// TwinCAT 3 PLC project MAIN
// ProgramVersion: 3.1.4024.0
// CompilerDefines: VISU_USEWSTRING
// libraries:
//   VisuElemMeter, * (System)
//   Tc2_EtherCAT, * (Beckhoff Automation GmbH)
//   Tc2_ModbusRTU, * (Beckhoff Automation GmbH)
//   Tc2_Standard, * (Beckhoff Automation GmbH)
//   Tc2_SUPS, * (Beckhoff Automation GmbH)
//   Tc2_System, * (Beckhoff Automation GmbH)
//   Tc2_Utilities, * (Beckhoff Automation GmbH)
//   Tc3_EventLogger, * (Beckhoff Automation GmbH)
//   Tc3_Module, * (Beckhoff Automation GmbH)
//   VisuDialogs, * (System)
// project tree:
//   DUTs/ ST_4Bytes.TcDUT, ST_Error.TcDUT, U_4Bytes2Real.TcDUT
//   / GlobalTextList.TcGTLO, ImagePool.TcIPO (not stored), PlcTask.TcTTO, PlcTask2.TcTTO, RecipeManager.TcRMO (not stored), Visualization Manager.TcVMO (not stored), VISU_TASK.TcTTO
//   GVLs/ GVL.TcGVL, GVL_ADS.TcGVL, GVL_HMI.TcGVL, GVL_IO.TcGVL, GVL_IoT.TcGVL, GVL_OF_VU.TcGVL, GVL_Retain.TcGVL
//   POUs/Components/Child Components/ FB_Conveyor.TcPOU, FB_Cylinder.TcPOU, FB_Interface_EtherCat.TcPOU, FB_Interface_MbRtu.TcPOU, FB_Inverter.TcPOU, FB_Loadcell.TcPOU, FB_SuctionCup.TcPOU
//   POUs/Components/Interfaces/ I_Conveyor.TcIO, I_Cylinder.TcIO, I_Inverter.TcIO, I_LoadCell.TcIO, I_SuctionCup.TcIO
//   POUs/Components/Sim Components/ FB_Conveyor_Sim.TcPOU, FB_Cylinder_Sim.TcPOU, FB_Inverter_Sim.TcPOU, FB_LoadCell_Sim.TcPOU, FB_SuctionCup_Sim.TcPOU
//   POUs/Functions/ FB_EventButton.TcPOU, FB_Eventlogger.TcPOU, F_SetError.TcPOU, F_SetWarning.TcPOU
//   POUs/Machines/ PR_Conveyor_Out.TcPOU, PR_Line01.TcPOU, PR_Line02.TcPOU
//   POUs/ MAIN.TcPOU, MAIN_LINE2.TcPOU
//   POUs/Modules/ FB_CupSupplyModule.TcPOU, FB_FoodMixerModule.TcPOU, FB_FoodWeightModule.TcPOU, FB_LidCloseModule.TcPOU, FB_LidSupplyModule.TcPOU, FB_Transfer.TcPOU, FB_WormWeightModule.TcPOU
//   POUs/Recipe/ PRG_MainRecipe1.TcPOU, PRG_MainRecipe1_1.TcPOU, PRG_RecipeList1.TcPOU, PRG_RecipeList1_1.TcPOU
//   VISUs/Alarm/ N_Alarm.TcVIS, N_Alarm_1.TcVIS
//   VISUs/IO/ N_Parameter_1.TcVIS, N_Parameter_2.TcVIS, N_PLC_I1.TcVIS, N_PLC_I1_next.TcVIS, N_PLC_I2.TcVIS, N_PLC_I2_next.TcVIS, N_PLC_O1.TcVIS, N_PLC_O2.TcVIS
//   VISUs/Main_Line/ MAIN_LINE1.TcVIS, MAIN_LINE2.TcVIS
//   VISUs/Manual/Line1/ N_FoodSupply1.TcVIS, N_JarSupply1.TcVIS, N_LidPressing1.TcVIS, N_LidSupply1.TcVIS, N_Tranfer1.TcVIS, N_WormWeight1.TcVIS
//   VISUs/Manual/Line2/ N_FoodSupply2.TcVIS, N_JarSupply2.TcVIS, N_LidPressing2.TcVIS, N_LidSupply2.TcVIS, N_Tranfer2.TcVIS, N_WormWeight2.TcVIS
//   VISUs/Recipe/ N_Recipe_Line1.TcVIS, N_Recipe_Line2.TcVIS
//   VISUs/Setting/ N_Setting_Delay_FoodSupply1.TcVIS, N_Setting_Delay_FoodSupply2.TcVIS, N_Setting_Delay_JarSupply1.TcVIS, N_Setting_Delay_JarSupply2.TcVIS, N_Setting_Delay_LidPressing1.TcVIS, N_Setting_Delay_LidPressing2.TcVIS, N_Setting_Delay_LidSupply1.TcVIS, N_Setting_Delay_LidSupply2.TcVIS, N_Setting_Delay_Tranfer1.TcVIS, N_Setting_Delay_Tranfer2.TcVIS, N_Setting_Delay_WormWeight1.TcVIS, N_Setting_Delay_WorwWeight2.TcVIS, N_Setting_Line1.TcVIS, N_Setting_Line2.TcVIS
//   VISUs/Title/ N_Footer_Alarm.TcVIS, N_Footer_Alarm_1.TcVIS, N_Footer_Line1.TcVIS, N_Footer_Line2.TcVIS, N_Header.TcVIS, N_Login.TcVIS, startpage.TcVIS
// real-time tasks:
//   TASK PlcTask: cycle T#10ms, priority 20, ADS port 350
//   TASK VISU_TASK: cycle T#10ms, priority 30, ADS port 351
//   TASK PlcTask2: cycle T#10ms, priority 21, ADS port 352
//   TASK VISU_TASK1: cycle T#10ms, priority 1, ADS port 353
// I/O:
//   DEVICE Device 1 (EtherCAT) (disabled), AmsNetId 192.168.1.12.2.1
//     Term 1 (EK1200) [EK1200-5000 EtherCAT Power supply (2A E-Bus)]
//       Term 2 (EL1008) [EL1008 8Ch. Dig. Input 24V, 3ms]
//       Term 3 (EL1008) [EL1008 8Ch. Dig. Input 24V, 3ms]
//       Term 4 (EL1008) [EL1008 8Ch. Dig. Input 24V, 3ms]
//       Term 5 (EL1008) [EL1008 8Ch. Dig. Input 24V, 3ms]
//       Term 6 (EL1008) [EL1008 8Ch. Dig. Input 24V, 3ms]
//       Term 7 (EL1008) [EL1008 8Ch. Dig. Input 24V, 3ms]
//       Term 8 (EL1819) [EL1819 16Ch. Dig. Input 24V, 10µs]
//       Term 9 (EL2809) [EL2809 16Ch. Dig. Output 24V, 0.5A]
//       Term 10 (EL2809) [EL2809 16Ch. Dig. Output 24V, 0.5A]
//       Term 11 (EL2809-0015) [EL2809-0015 16Ch. Dig. Output 24V DC, 0.35A, not short-circuit proof]
//       Term 12 (EL6021) [EL6021 Interface (RS422/485)]
//       Term 13 (EK1110) [EK1110 EtherCAT extension]
//     Box 14 (TLBETHERCAT) [TLBETHERCAT]
//     Box 15 (TLBETHERCAT) [TLBETHERCAT]
//     Box 16 (IND360) [IND360 ECS]
//     Box 17 (IND360) [IND360 ECS]
//   DEVICE Device 3 (NOV-DP-RAM) (disabled)
// variable links:
//   MAIN/MAIN Instance <-> Device 1 (EtherCAT)/Box 14 (TLBETHERCAT)
//     PlcTask2 Inputs/PR_Line02.fb_WormWeight.fbLoadcell.fbInterface.StatusLaumas1 <-> TxPDO/1 Byte In (13)
//     PlcTask2 Inputs/PR_Line02.fb_WormWeight.fbLoadcell.fbInterface.StatusLaumas2 <-> TxPDO/1 Byte In (12)
//     PlcTask2 Inputs/PR_Line02.fb_WormWeight.fbLoadcell.fbInterface.WeightLaumas1 <-> TxPDO/1 Byte In (3)
//     PlcTask2 Inputs/PR_Line02.fb_WormWeight.fbLoadcell.fbInterface.WeightLaumas2 <-> TxPDO/1 Byte In (2)
//     PlcTask2 Inputs/PR_Line02.fb_WormWeight.fbLoadcell.fbInterface.WeightLaumas3 <-> TxPDO/1 Byte In (1)
//     PlcTask2 Inputs/PR_Line02.fb_WormWeight.fbLoadcell.fbInterface.WeightLaumas4 <-> TxPDO/1 Byte In (0)
//     PlcTask2 Outputs/PR_Line02.fb_WormWeight.fbLoadcell.fbInterface.CMDLaumas <-> RxPDO/1 Byte Out (1)
//   MAIN/MAIN Instance <-> Device 1 (EtherCAT)/Box 15 (TLBETHERCAT)
//     PlcTask2 Inputs/PR_Line02.fb_FoodWeight.fbLoadcell.fbInterface.StatusLaumas1 <-> TxPDO/1 Byte In (13)
//     PlcTask2 Inputs/PR_Line02.fb_FoodWeight.fbLoadcell.fbInterface.StatusLaumas2 <-> TxPDO/1 Byte In (12)
//     PlcTask2 Inputs/PR_Line02.fb_FoodWeight.fbLoadcell.fbInterface.WeightLaumas1 <-> TxPDO/1 Byte In (3)
//     PlcTask2 Inputs/PR_Line02.fb_FoodWeight.fbLoadcell.fbInterface.WeightLaumas2 <-> TxPDO/1 Byte In (2)
//     PlcTask2 Inputs/PR_Line02.fb_FoodWeight.fbLoadcell.fbInterface.WeightLaumas3 <-> TxPDO/1 Byte In (1)
//     PlcTask2 Inputs/PR_Line02.fb_FoodWeight.fbLoadcell.fbInterface.WeightLaumas4 <-> TxPDO/1 Byte In (0)
//     PlcTask2 Outputs/PR_Line02.fb_FoodWeight.fbLoadcell.fbInterface.CMDLaumas <-> RxPDO/1 Byte Out (1)
//   MAIN/MAIN Instance <-> Device 1 (EtherCAT)/Box 16 (IND360)
//     PlcTask Inputs/PR_Line01.fb_WormWeight.fbLoadcell.fbInterface.IND_M_RD_Float <-> TxPDO-2Block/MB1 Requested Measuring Value
//     PlcTask Inputs/PR_Line01.fb_WormWeight.fbLoadcell.fbInterface.IND_M_RD_Response <-> TxPDO-2Block/MB1 Response
//     PlcTask Inputs/PR_Line01.fb_WormWeight.fbLoadcell.fbInterface.IND_M_RD_Status <-> TxPDO-2Block/MB1 Scale Status
//     PlcTask Inputs/PR_Line01.fb_WormWeight.fbLoadcell.fbInterface.IND_SB_STT1 <-> TxPDO-2Block/SB1 Status Group 1
//     PlcTask Inputs/PR_Line01.fb_WormWeight.fbLoadcell.fbInterface.IND_SB_STT2 <-> TxPDO-2Block/SB1 Status Group 2
//     PlcTask Inputs/PR_Line01.fb_WormWeight.fbLoadcell.fbInterface.IND_SB_STT3 <-> TxPDO-2Block/SB1 Status Group 3
//     PlcTask Outputs/PR_Line01.fb_WormWeight.fbLoadcell.fbInterface.IND_M_WR_Command <-> RxPDO-2Block/MB1 Command
//     PlcTask Outputs/PR_Line01.fb_WormWeight.fbLoadcell.fbInterface.IND_M_WR_Float <-> RxPDO-2Block/MB1 Command Value
//   MAIN/MAIN Instance <-> Device 1 (EtherCAT)/Box 17 (IND360)
//     PlcTask Inputs/PR_Line01.fb_FoodWeight.fbLoadcell.fbInterface.IND_M_RD_Float <-> TxPDO-2Block/MB1 Requested Measuring Value
//     PlcTask Inputs/PR_Line01.fb_FoodWeight.fbLoadcell.fbInterface.IND_M_RD_Response <-> TxPDO-2Block/MB1 Response
//     PlcTask Inputs/PR_Line01.fb_FoodWeight.fbLoadcell.fbInterface.IND_M_RD_Status <-> TxPDO-2Block/MB1 Scale Status
//     PlcTask Inputs/PR_Line01.fb_FoodWeight.fbLoadcell.fbInterface.IND_SB_STT1 <-> TxPDO-2Block/SB1 Status Group 1
//     PlcTask Inputs/PR_Line01.fb_FoodWeight.fbLoadcell.fbInterface.IND_SB_STT2 <-> TxPDO-2Block/SB1 Status Group 2
//     PlcTask Inputs/PR_Line01.fb_FoodWeight.fbLoadcell.fbInterface.IND_SB_STT3 <-> TxPDO-2Block/SB1 Status Group 3
//     PlcTask Outputs/PR_Line01.fb_FoodWeight.fbLoadcell.fbInterface.IND_M_WR_Command <-> RxPDO-2Block/MB1 Command
//     PlcTask Outputs/PR_Line01.fb_FoodWeight.fbLoadcell.fbInterface.IND_M_WR_Float <-> RxPDO-2Block/MB1 Command Value
//   MAIN/MAIN Instance <-> Device 1 (EtherCAT)/Term 1 (EK1200)/Term 10 (EL2809)
//     PlcTask Outputs/PR_Line01.fb_CupSupply.fbCylinder_Dw.bMoveRetract <-> Channel 9/Output
//     PlcTask Outputs/PR_Line01.fb_CupSupply.fbCylinder_Suction.bMoveRetract <-> Channel 14/Output
//     PlcTask Outputs/PR_Line01.fb_CupSupply.fbCylinder_Up.bMoveExtend <-> Channel 8/Output
//     PlcTask Outputs/PR_Line01.fb_LidClose.fbCylinder_LidClose.bMoveExtend <-> Channel 15/Output
//     PlcTask Outputs/PR_Line01.fb_LidSupply.fbCylinder_LidStopper.bMoveRetract <-> Channel 11/Output
//     PlcTask Outputs/PR_Line01.fb_LidSupply.fbCylinder_Suction.bMoveExtend <-> Channel 12/Output
//     PlcTask Outputs/PR_Line01.fb_LidSupply.fbLidSuctionValve.bSuck <-> Channel 13/Output
//     PlcTask Outputs/PR_Line01.fb_Transfer.fbCylinder_Clip.bMoveRetract <-> Channel 16/Output
//     PlcTask Outputs/PR_Line01.fb_WormWeight.fbCylinder.bMoveRetract <-> Channel 10/Output
//     PlcTask2 Outputs/PR_Line02.fb_CupSupply.fbCylinder_Suction.bMoveRetract <-> Channel 3/Output
//     PlcTask2 Outputs/PR_Line02.fb_LidClose.fbCylinder_LidClose.bMoveExtend <-> Channel 4/Output
//     PlcTask2 Outputs/PR_Line02.fb_LidSupply.fbCylinder_Suction.bMoveExtend <-> Channel 1/Output
//     PlcTask2 Outputs/PR_Line02.fb_LidSupply.fbLidSuctionValve.bSuck <-> Channel 2/Output
//     PlcTask2 Outputs/PR_Line02.fb_Transfer.fbCylinder_Clip.bMoveRetract <-> Channel 5/Output
//     PlcTask2 Outputs/PR_Line02.fb_Transfer.fbCylinder_Comb.bMoveExtend <-> Channel 6/Output
//     PlcTask2 Outputs/PR_Line02.fb_Transfer.fbCylinder_Move_Comb.bMoveExtend <-> Channel 7/Output
//   MAIN/MAIN Instance <-> Device 1 (EtherCAT)/Term 1 (EK1200)/Term 11 (EL2809-0015)
//     PlcTask Outputs/PR_Line01.fb_FoodMixer.fbInverter.bReverse <-> Channel 3/Output
//     PlcTask Outputs/PR_Line01.fb_FoodWeight.fbDriver.bReverse <-> Channel 6/Output
//     PlcTask Outputs/PR_Line01.fb_Transfer.fbCylinder_Comb.bMoveExtend <-> Channel 1/Output
//     PlcTask Outputs/PR_Line01.fb_Transfer.fbCylinder_Move_Comb.bMoveExtend <-> Channel 2/Output
//     PlcTask2 Outputs/PR_Line02.fb_FoodMixer.fbInverter.bReverse <-> Channel 4/Output
//     PlcTask2 Outputs/PR_Line02.fb_FoodWeight.fbDriver.bReverse <-> Channel 5/Output
//   MAIN/MAIN Instance <-> Device 1 (EtherCAT)/Term 1 (EK1200)/Term 12 (EL6021)
//     PlcTask Inputs/GVL.fbModbus.InData/D[{0..21}] <-> COM TxPDO-Map Inputs/Data In {0..21}  (22 links)
//     PlcTask Inputs/GVL.fbModbus.InData/Status <-> COM TxPDO-Map Inputs/Status
//     PlcTask Outputs/GVL.fbModbus.OutData/Ctrl <-> COM RxPDO-Map Outputs/Ctrl
//     PlcTask Outputs/GVL.fbModbus.OutData/D[{0..21}] <-> COM RxPDO-Map Outputs/Data Out {0..21}  (22 links)
//   MAIN/MAIN Instance <-> Device 1 (EtherCAT)/Term 1 (EK1200)/Term 2 (EL1008)
//     PlcTask Inputs/GVL_IO.bEmer <-> Channel 4/Input
//     PlcTask Inputs/GVL_IO.bReset <-> Channel 3/Input
//     PlcTask Inputs/GVL_IO.bStart <-> Channel 1/Input
//     PlcTask Inputs/GVL_IO.bStop <-> Channel 2/Input
//     PlcTask Inputs/PR_Conveyor_Out.fb_Conveyor.bError_Motor_Mixer <-> Channel 7/Input
//     PlcTask Inputs/PR_Line01.fb_FoodMixer.bError_Motor_Mixer <-> Channel 8/Input
//     PlcTask2 Inputs/PR_Line02.fb_FoodMixer.bError_Motor_Mixer <-> Channel 5/Input
//     PlcTask2 Inputs/PR_Line02.fb_WormWeight.bError_Inverter <-> Channel 6/Input
//   MAIN/MAIN Instance <-> Device 1 (EtherCAT)/Term 1 (EK1200)/Term 3 (EL1008)
//     PlcTask Inputs/PR_Line01.fb_FoodWeight.bError_Driver <-> Channel 3/Input
//     PlcTask Inputs/PR_Line01.fb_WormWeight.bError_Inverter <-> Channel 1/Input
//     PlcTask2 Inputs/PR_Line02.fb_CupSupply.bCupDrop <-> Channel 8/Input
//     PlcTask2 Inputs/PR_Line02.fb_CupSupply.bCupEmpty <-> Channel 4/Input
//     PlcTask2 Inputs/PR_Line02.fb_CupSupply.fbCylinder_Dw.bAtExtend <-> Channel 7/Input
//     PlcTask2 Inputs/PR_Line02.fb_CupSupply.fbCylinder_Dw.bAtRetract <-> Channel 6/Input
//     PlcTask2 Inputs/PR_Line02.fb_CupSupply.fbCylinder_Up.bAtRetract <-> Channel 5/Input
//     PlcTask2 Inputs/PR_Line02.fb_FoodWeight.bError_Driver <-> Channel 2/Input
//   MAIN/MAIN Instance <-> Device 1 (EtherCAT)/Term 1 (EK1200)/Term 4 (EL1008)
//     PlcTask2 Inputs/PR_Line02.fb_LidClose.fbCylinder_LidClose.bAtRetract <-> Channel 8/Input
//     PlcTask2 Inputs/PR_Line02.fb_LidSupply.bLidEmpty <-> Channel 2/Input
//     PlcTask2 Inputs/PR_Line02.fb_LidSupply.fbCylinder_LidStopper.bAtExtend <-> Channel 4/Input
//     PlcTask2 Inputs/PR_Line02.fb_LidSupply.fbCylinder_LidStopper.bAtRetract <-> Channel 3/Input
//     PlcTask2 Inputs/PR_Line02.fb_LidSupply.fbCylinder_Suction.bAtExtend <-> Channel 6/Input
//     PlcTask2 Inputs/PR_Line02.fb_LidSupply.fbCylinder_Suction.bAtRetract <-> Channel 5/Input
//     PlcTask2 Inputs/PR_Line02.fb_LidSupply.fbLidSuctionValve.bPressure <-> Channel 7/Input
//     PlcTask2 Inputs/PR_Line02.fb_WormWeight.fbCylinder.bAtRetract <-> Channel 1/Input
//   MAIN/MAIN Instance <-> Device 1 (EtherCAT)/Term 1 (EK1200)/Term 5 (EL1008)
//     PlcTask2 Inputs/PR_Line02.fb_FoodWeight.bCupPresent <-> Channel 8/Input
//     PlcTask2 Inputs/PR_Line02.fb_LidClose.fbCylinder_LidClose.bAtExtend <-> Channel 1/Input
//     PlcTask2 Inputs/PR_Line02.fb_Transfer.fbCylinder_Clip.bAtExtend <-> Channel 7/Input
//     PlcTask2 Inputs/PR_Line02.fb_Transfer.fbCylinder_Clip.bAtRetract <-> Channel 6/Input
//     PlcTask2 Inputs/PR_Line02.fb_Transfer.fbCylinder_Comb.bAtExtend <-> Channel 3/Input
//     PlcTask2 Inputs/PR_Line02.fb_Transfer.fbCylinder_Comb.bAtRetract <-> Channel 2/Input
//     PlcTask2 Inputs/PR_Line02.fb_Transfer.fbCylinder_Move_Comb.bAtExtend <-> Channel 5/Input
//     PlcTask2 Inputs/PR_Line02.fb_Transfer.fbCylinder_Move_Comb.bAtRetract <-> Channel 4/Input
//   MAIN/MAIN Instance <-> Device 1 (EtherCAT)/Term 1 (EK1200)/Term 6 (EL1008)
//     PlcTask Inputs/PR_Line01.fb_CupSupply.bCupDrop <-> Channel 6/Input
//     PlcTask Inputs/PR_Line01.fb_CupSupply.bCupEmpty <-> Channel 2/Input
//     PlcTask Inputs/PR_Line01.fb_CupSupply.fbCylinder_Dw.bAtExtend <-> Channel 5/Input
//     PlcTask Inputs/PR_Line01.fb_CupSupply.fbCylinder_Dw.bAtRetract <-> Channel 4/Input
//     PlcTask Inputs/PR_Line01.fb_CupSupply.fbCylinder_Up.bAtRetract <-> Channel 3/Input
//     PlcTask Inputs/PR_Line01.fb_LidSupply.bLidEmpty <-> Channel 8/Input
//     PlcTask Inputs/PR_Line01.fb_WormWeight.fbCylinder.bAtRetract <-> Channel 7/Input
//     PlcTask2 Inputs/PR_Line02.fb_WormWeight.bCupPresent <-> Channel 1/Input
//   MAIN/MAIN Instance <-> Device 1 (EtherCAT)/Term 1 (EK1200)/Term 7 (EL1008)
//     PlcTask Inputs/PR_Line01.fb_LidClose.fbCylinder_LidClose.bAtExtend <-> Channel 7/Input
//     PlcTask Inputs/PR_Line01.fb_LidClose.fbCylinder_LidClose.bAtRetract <-> Channel 6/Input
//     PlcTask Inputs/PR_Line01.fb_LidSupply.fbCylinder_LidStopper.bAtExtend <-> Channel 2/Input
//     PlcTask Inputs/PR_Line01.fb_LidSupply.fbCylinder_LidStopper.bAtRetract <-> Channel 1/Input
//     PlcTask Inputs/PR_Line01.fb_LidSupply.fbCylinder_Suction.bAtExtend <-> Channel 4/Input
//     PlcTask Inputs/PR_Line01.fb_LidSupply.fbCylinder_Suction.bAtRetract <-> Channel 3/Input
//     PlcTask Inputs/PR_Line01.fb_LidSupply.fbLidSuctionValve.bPressure <-> Channel 5/Input
//     PlcTask Inputs/PR_Line01.fb_Transfer.fbCylinder_Comb.bAtRetract <-> Channel 8/Input
//   MAIN/MAIN Instance <-> Device 1 (EtherCAT)/Term 1 (EK1200)/Term 8 (EL1819)
//     PlcTask Inputs/GVL_IO.bCheckVan <-> Channel 13/Input
//     PlcTask Inputs/GVL_IO.bSafetyDoor1 <-> Channel 9/Input
//     PlcTask Inputs/GVL_IO.bSafetyDoor2 <-> Channel 8/Input
//     PlcTask Inputs/GVL_IO.bSafetyDoor3 <-> Channel 10/Input
//     PlcTask Inputs/PR_Line01.fb_CupSupply.fbCylinder_Suction.bAtExtend <-> Channel 11/Input
//     PlcTask Inputs/PR_Line01.fb_FoodWeight.bCupPresent <-> Channel 6/Input
//     PlcTask Inputs/PR_Line01.fb_Transfer.fbCylinder_Clip.bAtExtend <-> Channel 5/Input
//     PlcTask Inputs/PR_Line01.fb_Transfer.fbCylinder_Clip.bAtRetract <-> Channel 4/Input
//     PlcTask Inputs/PR_Line01.fb_Transfer.fbCylinder_Comb.bAtExtend <-> Channel 1/Input
//     PlcTask Inputs/PR_Line01.fb_Transfer.fbCylinder_Move_Comb.bAtExtend <-> Channel 3/Input
//     PlcTask Inputs/PR_Line01.fb_Transfer.fbCylinder_Move_Comb.bAtRetract <-> Channel 2/Input
//     PlcTask Inputs/PR_Line01.fb_WormWeight.bCupPresent <-> Channel 7/Input
//     PlcTask2 Inputs/PR_Line02.fb_CupSupply.fbCylinder_Suction.bAtExtend <-> Channel 12/Input
//   MAIN/MAIN Instance <-> Device 1 (EtherCAT)/Term 1 (EK1200)/Term 9 (EL2809)
//     PlcTask Outputs/GVL_IO.bLight_Running <-> Channel 1/Output
//     PlcTask Outputs/GVL_IO.bLight_Stop <-> Channel 2/Output
//     PlcTask Outputs/GVL_IO.bSirens <-> Channel 8/Output
//     PlcTask Outputs/PR_Conveyor_Out.fb_Conveyor.fbInverter.bVFD <-> Channel 5/Output
//     PlcTask Outputs/PR_Line01.fb_FoodMixer.fbInverter.bVFD <-> Channel 6/Output
//     PlcTask Outputs/PR_Line01.fb_FoodWeight.fbDriver.bReset <-> Channel 11/Output
//     PlcTask Outputs/PR_Line01.fb_FoodWeight.fbDriver.bVFD <-> Channel 12/Output
//     PlcTask Outputs/PR_Line01.fb_WormWeight.fbInverter.bVFD <-> Channel 7/Output
//     PlcTask2 Outputs/PR_Line02.fb_CupSupply.fbCylinder_Dw.bMoveRetract <-> Channel 14/Output
//     PlcTask2 Outputs/PR_Line02.fb_CupSupply.fbCylinder_Up.bMoveExtend <-> Channel 13/Output
//     PlcTask2 Outputs/PR_Line02.fb_FoodMixer.fbInverter.bVFD <-> Channel 3/Output
//     PlcTask2 Outputs/PR_Line02.fb_FoodWeight.fbDriver.bReset <-> Channel 9/Output
//     PlcTask2 Outputs/PR_Line02.fb_FoodWeight.fbDriver.bVFD <-> Channel 10/Output
//     PlcTask2 Outputs/PR_Line02.fb_LidSupply.fbCylinder_LidStopper.bMoveRetract <-> Channel 16/Output
//     PlcTask2 Outputs/PR_Line02.fb_WormWeight.fbCylinder.bMoveRetract <-> Channel 15/Output
//     PlcTask2 Outputs/PR_Line02.fb_WormWeight.fbInverter.bVFD <-> Channel 4/Output

CONFIGURATION MAIN
    RESOURCE PLC ON TwinCAT3
        TASK PlcTask(INTERVAL := T#10ms, PRIORITY := 20);
        TASK PlcTask2(INTERVAL := T#10ms, PRIORITY := 21);
        TASK VISU_TASK(INTERVAL := T#10ms, PRIORITY := 1);
        PROGRAM MAIN WITH PlcTask : MAIN;
        PROGRAM MAIN_LINE2 WITH PlcTask2 : MAIN_LINE2;
        PROGRAM VisuElems_Visu_Prg WITH VISU_TASK : VisuElems.Visu_Prg;
    END_RESOURCE
END_CONFIGURATION

// ---- DUTs/ST_4Bytes.TcDUT
TYPE ST_4Bytes :
STRUCT
	Byte1	: BYTE;
	Byte2	: BYTE;
	Byte3	: BYTE;
	Byte4	: BYTE;
END_STRUCT
END_TYPE

// ---- DUTs/ST_Error.TcDUT
TYPE ST_Error :
STRUCT
	nErrorID  	: INT;
	ErrorTime 	: DT;
	ErrorStatus : BOOL;
END_STRUCT
END_TYPE

// ---- DUTs/U_4Bytes2Real.TcDUT
TYPE U_4Bytes2Real :
UNION
	fReal	: DINT;
	st4bytes: ST_4Bytes;
END_UNION
END_TYPE

// ---- GVLs/GVL.TcGVL
VAR_GLOBAL
	bSimMode			: BOOL;
	// var sim Inverter with Loadcell
	bHaveLoad			: BOOL; // run inverter = true
	fInvSpeed			: REAL;
	//Error system
	bError1				: BOOL;
	bError2				: BOOL;
	nErrorID			: INT;
	stErrorTxt			: WSTRING;
	stErrorTxt1			: STRING;
	stErrorTxt2			: WSTRING;
	stErrorTxt3			: STRING;
	bWarning			: BOOL;
	bWarning2			: BOOL;
	nWarningID			: INT;
	stWarningTxt		: WSTRING;
	stWarningTxt1		: STRING;
	stWarningTxt2		: WSTRING;
	StWarningTxt3		: STRING;
	fbModbus			: ModbusRtuMaster_KL6x22B;
	bStartLine1			: BOOL;
	bStartLine2			: BOOL;
	SystemTimeFull 		: STRING;
	WritePSData			: WritePersistentData;
	bWriteData			: BOOL;
	t					: BYTE := 1;
	bToDropcup1			: BOOL;
	bToDropcup2			: BOOL;
	Run_conveyor		: R_TRIG;
	bRun				: BOOL;
	bRunAuto			: BOOL;
	bStopConv			: BOOL;
	Stop_conveyor		: R_TRIG;
	bResetmanual1		: BOOL;
	bResetmanual2		: BOOL;
	bResetAuto1			: BOOL;
	bResetAuto2			: BOOL;
	bfinish1			: BOOL;
	bfinish2			: BOOL;
	openstartpage		: BOOL;
	getuser				: STRING;
	GetLocalSystemTime 	: FB_LocalSystemTime;
	bWrn				: BOOL;
	bWrn2				: BOOL;
	bAlarm_Iot			: BOOL;
	bxoa				: BOOL;
	bTo_alarm_side		: BOOL;
	bTo_alarm_side2		: BOOL;
	Onlyday				: STRING;
	OnlyTime			: STRING;
	bclearall			: BOOL;
	button				: ARRAY [1..40] OF BOOL;
	//change line 1
	fFast_Speed_line1_change						: REAL;//FoodWeight
	fSlow_Speed_1_line1_change						: REAL;
	fSlow_Speed_2_line1_change						: REAL;
	fDerisedWeight_Food_line1_change				: REAL;
	fChangeMode_Food_1_line1_change					: REAL;
	fChangeMode_Food_2_line1_change					: REAL;
	fPerStop_Food_line1_change						: REAL;
	fTimer_Check_Food_line1_change					: REAL;
	fDelta_Food_line1_change						: REAL;
	fFast_Speed_vibrating_funnel_line1_change		: REAL;//WormWeight
	fSlow_Speed_vibrating_funnel_1_line1_change		: REAL;
	fSlow_Speed_vibrating_funnel_2_line1_change		: REAL;
	fDerisedWeight_Worm_line1_change				: REAL;
	fChangeMode_Worm_1_line1_change					: REAL;
	fChangeMode_Worm_2_line1_change					: REAL;
	fPerStop_Worm_line1_change						: REAL;
	fTimer_Check_Worm_line1_change					: REAL;
	fDelta_Worm_line1_change						: REAL;
	//change line 2
	fFast_Speed_line2_change						: REAL;//FoodWeight
	fSlow_Speed_1_line2_change						: REAL;
	fSlow_Speed_2_line2_change						: REAL;
	fDerisedWeight_Food_line2_change				: REAL;
	fChangeMode_Food_1_line2_change					: REAL;
	fChangeMode_Food_2_line2_change					: REAL;
	fPerStop_Food_line2_change						: REAL;
	fTimer_Check_Food_line2_change					: REAL;
	fDelta_Food_line2_change						: REAL;
	fFast_Speed_vibrating_funnel_line2_change		: REAL;//WormWeight
	fSlow_Speed_vibrating_funnel_1_line2_change		: REAL;
	fSlow_Speed_vibrating_funnel_2_line2_change		: REAL;
	fDerisedWeight_Worm_line2_change				: REAL;
	fChangeMode_Worm_1_line2_change					: REAL;
	fChangeMode_Worm_2_line2_change					: REAL;
	fPerStop_Worm_line2_change						: REAL;
	fTimer_Check_Worm_line2_change					: REAL;
	fDelta_Worm_line2_change						: REAL;
END_VAR

// ---- GVLs/GVL_ADS.TcGVL
VAR_GLOBAL
END_VAR

// ---- GVLs/GVL_HMI.TcGVL
VAR_GLOBAL 
	//system
	hienthiDialog		: BOOL;
	hienthiDialog2		: BOOL;
	bResetErr1			: BOOL;
	bStart1				: BOOL;
	bStart2				: BOOL;
	bStop1				: BOOL;
	bStop2				: BOOL;
	bShift_is_over1		: BOOL;
	bShift_is_over2		: BOOL;
	bResetErr2			: BOOL;
	bStatusStart1		: BOOL;
	bStatusStart2		: BOOL;
	Busy				: ARRAY [1..7] OF BOOL;
	Error				: ARRAY [1..7] OF BOOL;
	ErrorID				: ARRAY [1..7] OF MODBUS_ERRORS;
	bSave1				: BOOL;
	bLoad1				: BOOL;
	bDelete1			: BOOL;
	nStatus1			: STRING;
	nStatus2			: STRING;
	bClear1				: BOOL;
	bClear2				: BOOL;
	bypass				: BOOL;
	hienthibypass		: BOOL;
	bSave2				: BOOL;
	bLoad2				: BOOL;
	bDelete2			: BOOL;
	AlarmList 			: ARRAY [1..4, 1..100] OF WSTRING;
	AlarmList2 			: ARRAY [1..4, 1..100] OF WSTRING;
	AlarmList3			: ARRAY [1..4, 1..100] OF STRING;
	AlarmList4			: ARRAY [1..4, 1..100] OF STRING;
END_VAR

// ---- GVLs/GVL_IO.TcGVL
VAR_GLOBAL
	bStart			AT %I* : BOOL;
	bStop			AT %I* : BOOL;
	bReset			AT %I* : BOOL;
	bEmer			AT %I* : BOOL;
	bSafetyDoor1	AT %I* : BOOL;
	bSafetyDoor2	AT %I* : BOOL;
	bSafetyDoor3	AT %I* : BOOL;
	bCheckVan		AT %I* : BOOL;
	bLight_Running 	AT %Q* : BOOL;
	bLight_Stop		AT %Q* : BOOL;
	bSirens			AT %Q* : BOOL;
END_VAR

// ---- GVLs/GVL_IoT.TcGVL
VAR_GLOBAL
	username					: STRING;
	fWeight_Food_line1			: REAL;
	fWeight_Worm_line1			: REAL;
	fDerisedWeight_Food_line1	: REAL;
	fDerisedWeight_Worm_line1	: REAL;
	fActDelta_Food_line1		: REAL;
	fActDelta_Worm_line1		: REAL;	
	fWeight_Food_line2			: REAL;
	fWeight_Worm_line2			: REAL;
	fDerisedWeight_Food_line2	: REAL;
	fDerisedWeight_Worm_line2	: REAL;
	fActDelta_Food_line2		: REAL;
	fActDelta_Worm_line2		: REAL;	
	Time_Start_Food_line1		: DT;
	Time_Stop_Food_line1		: DT;
	Time_Start_Worm_line1		: DT;
	Time_Stop_Worm_line1		: DT;	
	Time_Start_Food_line2		: DT;
	Time_Stop_Food_line2		: DT;
	Time_Start_Worm_line2		: DT;
	Time_Stop_Worm_line2		: DT;	
	status						: STRING;	
	fDelta_Food_line1			: REAL;
	fDelta_Worm_line1			: REAL;
	fDelta_Food_line2			: REAL;
	fDelta_Worm_line2			: REAL;
	bStatus_Food_line1			: STRING;
	bStatus_Worm_line1			: STRING;
	bStatus_Food_line2			: STRING;
	bStatus_Worm_line2			: STRING;
	bAlarm						: BOOL;
END_VAR

// ---- GVLs/GVL_OF_VU.TcGVL
VAR_GLOBAL
	bDeleteRecipe1  			: BOOL;
	bDeleteRecipe2				: BOOL;
	//////////////test////////////////////
	// vara for main line	////
	bVN							: BOOL;
	LineName					: ARRAY[1..2] OF INT;
	setLinet					: INT;
	bRunMachine					: ARRAY[1..2] OF BOOL;
	data_worm1 					: ARRAY[1..2] OF ARRAY[1..10] OF REAL;
	data_worm2					: ARRAY[1..2] OF ARRAY[1..10] OF REAL;
	Run 						: ARRAY[1..2] OF BOOL;
	sOperationStatus			: ARRAY[1..2] OF STRING := ['running','waiting'];
	fMassOfCup					: ARRAY[1..2] OF REAL := [35.05,56.36];
	fMassOfFoodAct				: ARRAY[1..2] OF REAL := [5.6,3.4];
	fMassOfFoodSet				: ARRAY[1..2] OF REAL := [5.6,3.0];
	fDeviationFoodAct			: ARRAY[1..2] OF REAL;
	fDeviationFoodSet			: ARRAY[1..2] OF REAL;
	fMassOfWormAct				: ARRAY[1..2] OF REAL := [10.5,8.3];
	fMassOfWormSet				: ARRAY[1..2] OF REAL := [9.6,8.3];
	fDeviationWormAct			: ARRAY[1..2] OF REAL;
	fDeviationWormSet			: ARRAY[1..2] OF REAL;
	bClear						: ARRAY[1..2] OF BOOL;
	bIsSuccessFood				: ARRAY[1..2] OF BOOL := [TRUE,FALSE];
	bIsSuccessWorm				: ARRAY[1..2] OF BOOL := [FALSE,TRUE];
	fWeightFood					: ARRAY[1..2] OF REAL;
	fWeightWorm					: ARRAY[1..2] OF REAL;

	// just add ///
	nSuccess					: ARRAY[1..2] OF INT :=[10,8];
	nFail						: ARRAY[1..2] OF INT :=[2,5];
	nCounter					: ARRAY[1..2] OF INT :=[12,13];
	fFlowWormMain				: ARRAY[1..2] OF REAL:=[9.56,8.34];
	fFlowFoodMain				: ARRAY[1..2] OF REAL:=[3.2,5.4];
	fDelayMain					: ARRAY[1..2] OF REAL:=[3,4];
	sNameRecipe					: ARRAY[1..2] OF STRING:=['recipe1', 'reccipe2'];
	
	///IO////
	bSensorOutOfLid				: ARRAY[1..2] OF BOOL := [FALSE,TRUE];
	bSensorOutOfJar				: ARRAY[1..2] OF BOOL := [FALSE,TRUE];
	bSensorReleaseJar			: ARRAY[1..2] OF BOOL := [TRUE,FALSE];
	bSensorJarInStation			: ARRAY[1..2] OF BOOL := [TRUE,FALSE];
	bSensorSuckLid				: ARRAY[1..2] OF BOOL := [FALSE,TRUE];
	bSensorDoor					: ARRAY[1..4] OF BOOL := [TRUE,FALSE];
	bUpperCylinderJar			: ARRAY[1..2] OF BOOL;
	bLowerCylinderJar			: ARRAY[1..2] OF BOOL;
	bAgitatiorMotor				: ARRAY[1..2] OF BOOL := [TRUE,FALSE];
	bDispenserMotor				: ARRAY[1..2] OF BOOL := [TRUE,FALSE];
	bVibrattingFunnel			: ARRAY[1..2] OF BOOL := [FALSE,TRUE];
	bOutputConveyor				: BOOL;
	bCylinderMoveComb			: ARRAY[1..2] OF BOOL := [TRUE,FALSE];
	bCylinderMoveCombInOut		: ARRAY[1..2] OF BOOL := [TRUE,FALSE];
	bCylinderClampJar			: ARRAY[1..2] OF BOOL := [TRUE,FALSE];
	bCylinderSuckReleaseLid		: ARRAY[1..2] OF BOOL := [TRUE,FALSE];
	bValveSuckLlid				: ARRAY[1..2] OF BOOL := [FALSE,TRUE];
	bCylinderBlockWorm			: ARRAY[1..2] OF BOOL := [TRUE,FALSE];
	bCylinderBlockLidRail		: ARRAY[1..2] OF BOOL := [TRUE,FALSE];
	bValveLocateJar				: ARRAY[1..2] OF BOOL := [FALSE,TRUE];
	bCylinderPressLid			: ARRAY[1..2] OF BOOL := [FALSE,TRUE];
	bHorn						: BOOL := TRUE;
	bStartLamp					: ARRAY[1..2] OF BOOL := [FALSE,TRUE];
	bStopLamp					: ARRAY[1..2] OF BOOL := [TRUE,FALSE];
	bValveBlowLid				: ARRAY[1..2] OF BOOL := [FALSE,TRUE];
	
	
	//Var for Weight Worm Cluster /////////////
	bRunVibratingFunnel			: ARRAY[1..2] OF BOOL;
	fFreqVibratingFunnel		: ARRAY[1..2] OF REAL;
	bAddFreqVibratingFunnel		: ARRAY[1..2] OF BOOL;
	bSubFreqVibratingFunnel		: ARRAY[1..2] OF BOOL;
	bRunCylinderBlockWormExt	: ARRAY[1..2] OF BOOL;
	bRunCylinderBlockWormRet	: ARRAY[1..2] OF BOOL;
	bSet0Worm					: ARRAY[1..2] OF BOOL;
	fWomrMassTotal				: ARRAY[1..2] OF REAL;
	fFlowWorm					: ARRAY[1..2] OF REAL;
	
	//Var for Lid Supply Cluster
	bRunValveSuckLid			: ARRAY[1..2] OF BOOL;
	bRunValveReleasekLid		: ARRAY[1..2] OF BOOL;
	bRunCylinderSuckReleaseLidExt: ARRAY[1..2] OF BOOL;
	bRunCylinderSuckReleaseLidRet: ARRAY[1..2] OF BOOL;
	bRunCylinderBlockLidRailExt	: ARRAY[1..2] OF BOOL;
	bRunCylinderBlockLidRailRet	: ARRAY[1..2] OF BOOL;
	
	//Var for Jar Supply Cluster
	bRunUpperCylinderBlockLidExt: ARRAY[1..2] OF BOOL;
	bRunUpperCylinderBlockLidRet: ARRAY[1..2] OF BOOL;
	bRunLowerCylinderBlockLidExt: ARRAY[1..2] OF BOOL;
	bRunLowerCylinderBlockLidRet: ARRAY[1..2] OF BOOL;
	
	//Var for Food Supply Cluster
	bRunAgitatorMotor			: ARRAY[1..2] OF BOOL;
	fFreqAgitatorMotor			: ARRAY[1..2] OF REAL;
	bAddFreqAgitatorMotor		: ARRAY[1..2] OF BOOL;
	bSubFreqAgitatorMotor		: ARRAY[1..2] OF BOOL;
	
	bRunDispenserMotor			: ARRAY[1..2] OF BOOL;
	fFreqDispenserMotor			: ARRAY[1..2] OF REAL;
	bAddFreqDispenserMotor		: ARRAY[1..2] OF BOOL;
	bSubFreqDispenserMotor		: ARRAY[1..2] OF BOOL;
	bSet0Food					: ARRAY[1..2] OF BOOL;
	fFoodMassTotal				: ARRAY[1..2] OF REAL;
	fFlowFood					: ARRAY[1..2] OF REAL;
	
	//Var for Pressing Lid Cluster
	bRunCylinderPressLidExt		: ARRAY[1..2] OF BOOL;
	bRunCylinderPressLidRet		: ARRAY[1..2] OF BOOL;
	bRunValveLocateJar			: ARRAY[1..2] OF BOOL;
	
	//Var for Transfer Cluster
	bRunCylinderMoveCombExt		: ARRAY[1..2] OF BOOL;
	bRunCylinderMoveCombRet		: ARRAY[1..2] OF BOOL;
	bRunCylinderMoveCombInOutExt: ARRAY[1..2] OF BOOL;
	bRunCylinderMoveCombInOutRet: ARRAY[1..2] OF BOOL;
	bRunCylinderClampCombJarExt	: ARRAY[1..2] OF BOOL;
	bRunCylinderClampCombJarRet	: ARRAY[1..2] OF BOOL;
	fFreqOutputConveyor			: REAL;
	bRunOutputConveyor			: BOOL;
	bAddFreqOutputConveyor		: BOOL;
	bSubFreqOutputConveyor		: BOOL;
	// Setting parameter ////
	fMassDesireFood				: ARRAY[1..2] OF REAL;
	fAllowableDeviationFood		: ARRAY[1..2] OF REAL;
	fSpeedIFood					: ARRAY[1..2] OF REAL;
	fSppedIIFood				: ARRAY[1..2] OF REAL;
	fSpeedIIIFood				: ARRAY[1..2] OF REAL;
	fChangeI_IIFood				: ARRAY[1..2] OF REAL;
	fChangeII_IIIFood			: ARRAY[1..2] OF REAL;
	fMaxPayLoadFood				: ARRAY[1..2] OF REAL;
	fPosHaltFood				: ARRAY[1..2] OF REAL;
	fDelayFood					: ARRAY[1..2] OF REAL;
	
	fMassDesireWorm				: ARRAY[1..2] OF REAL;
	fAllowableDeviationWorm		: ARRAY[1..2] OF REAL;
	fSpeedIWorm					: ARRAY[1..2] OF REAL;
	fSppedIIWorm				: ARRAY[1..2] OF REAL;
	fSpeedIIIWorm				: ARRAY[1..2] OF REAL;
	fChangeI_IIWorm				: ARRAY[1..2] OF REAL;
	fChangeII_IIIWorm			: ARRAY[1..2] OF REAL;
	fMaxPayLoadWorm				: ARRAY[1..2] OF REAL;
	fPosHaltWorm				: ARRAY[1..2] OF REAL;
	fDelayWorm					: ARRAY[1..2] OF REAL;
	
	// Recipe parametters ///
	fRecMassOfFood				: ARRAY[1..2] OF REAL;
	fRecMassOfWorm				: ARRAY[1..2] OF REAL;
	fRecDeviationOfFood			: ARRAY[1..2] OF REAL;
	fRecDeviationOfWorm			: ARRAY[1..2] OF REAL;
	fRecSpeedIOfFood			: ARRAY[1..2] OF REAL;
	fRecSpeedIOfWorm			: ARRAY[1..2] OF REAL;
	fRecSpeedIIOfFood			: ARRAY[1..2] OF REAL;
	fRecSpeedIIOfWorm			: ARRAY[1..2] OF REAL;
	fRecSpeedIIIOfFood			: ARRAY[1..2] OF REAL;
	fRecSpeedIIIOfWorm			: ARRAY[1..2] OF REAL;
	fRecChangeI_IIOfFood		: ARRAY[1..2] OF REAL;
	fRecChangeI_IIOfWorm		: ARRAY[1..2] OF REAL;
	fRecChangeII_IIIOfFood		: ARRAY[1..2] OF REAL;
	fRecChangeII_IIIOfWorm		: ARRAY[1..2] OF REAL;
	fRecMaxPayLoadOfFood		: ARRAY[1..2] OF REAL;
	fRecMaxPayLoadOfWorm		: ARRAY[1..2] OF REAL;
	fRecHaltPosOfFood			: ARRAY[1..2] OF REAL;
	fRecHaltPosOfWorm			: ARRAY[1..2] OF REAL;
	fRecDelayOfFood				: ARRAY[1..2] OF REAL;
	fRecDelayOfWorm				: ARRAY[1..2] OF REAL;
	bRecSave					: ARRAY[1..2] OF BOOL;
	bRecLoad					: ARRAY[1..2] OF BOOL;
	bRecDelete					: ARRAY[1..2] OF BOOL;
	GetFullTime					: STRING;
	GetDate						: STRING;	
	GetTime						: STRING;

	
		
	
END_VAR

// ---- GVLs/GVL_Retain.TcGVL
VAR_GLOBAL PERSISTENT
	nErrorIDList1		: ARRAY[1..100] OF ST_Error;
	nErrorIDList2		: ARRAY[1..100] OF ST_Error;
	a2 					: INT;
	i 					: INT := 1;
	nResult_true1		: INT;
	nResult_false1		: INT;
	nCount1				: INT;
	nResult_true2		: INT;
	nResult_false2		: INT;
	nCount2				: INT;
	nShoot1				: REAL;
	nShoot2				: REAL;
END_VAR

// ---- POUs/Components/Interfaces/I_Conveyor.TcIO
INTERFACE I_Conveyor

PROPERTY IsRun : BOOL
GET
END_GET
END_PROPERTY

METHOD Start : BOOL
VAR_INPUT
END_VAR
END_METHOD

METHOD Stop : BOOL
VAR_INPUT
END_VAR
END_METHOD

END_INTERFACE

// ---- POUs/Components/Interfaces/I_Cylinder.TcIO
INTERFACE I_Cylinder

PROPERTY bIsExtend : BOOL
GET
END_GET
END_PROPERTY

PROPERTY bIsRetract : BOOL
GET
END_GET
END_PROPERTY

METHOD Extend : BOOL
VAR_INPUT
END_VAR
END_METHOD

METHOD Retract : BOOL
VAR_INPUT
END_VAR
END_METHOD

END_INTERFACE

// ---- POUs/Components/Interfaces/I_Inverter.TcIO
INTERFACE I_Inverter

PROPERTY ActualSpeed : REAL
GET
END_GET
END_PROPERTY

PROPERTY bIsMove : BOOL
GET
END_GET
END_PROPERTY

PROPERTY fTargetSpeed : REAL
GET
END_GET
SET
END_SET
END_PROPERTY

METHOD Reset : BOOL
VAR_INPUT
END_VAR
END_METHOD

METHOD Reverse : BOOL
VAR_INPUT
END_VAR
END_METHOD

METHOD Start : BOOL
VAR_INPUT
END_VAR
END_METHOD

METHOD Stop : BOOL
VAR_INPUT
END_VAR
END_METHOD

END_INTERFACE

// ---- POUs/Components/Interfaces/I_LoadCell.TcIO
INTERFACE I_LoadCell

PROPERTY fActWeight : REAL
GET
END_GET
END_PROPERTY

METHOD NetMode : BOOL
VAR_INPUT
END_VAR
END_METHOD

METHOD Set_Zero : BOOL
VAR_INPUT
END_VAR
END_METHOD

PROPERTY Status : REAL
GET
END_GET
END_PROPERTY

END_INTERFACE

// ---- POUs/Components/Interfaces/I_SuctionCup.TcIO
INTERFACE I_SuctionCup

PROPERTY bIsSuck : BOOL
GET
END_GET
END_PROPERTY

PROPERTY fThreshold : REAL
GET
END_GET
SET
END_SET
END_PROPERTY

METHOD Release : BOOL
VAR_INPUT
END_VAR
END_METHOD

METHOD Suck : BOOL
VAR_INPUT
END_VAR
END_METHOD

END_INTERFACE

// ---- POUs/MAIN.TcPOU
PROGRAM MAIN
VAR
	traError			: BOOL;
	traInitDone			: BOOL;
	bModeOff			: BOOL;
	bModeManual			: BOOL := TRUE;
	bModeAuto			: BOOL;
	Err_T				: R_TRIG;
	Wrn_T				: R_TRIG;
	Wrn_T1				: R_TRIG;
	Reset_T				: R_TRIG;
	fbtimer				: TON;
	fbTimerSirens		: TON;
	fbTimer_IoT			: Ton;
	Run_T				: R_TRIG;
	Stop_T				: R_TRIG;
	k,k1				: INT;
	nState				: INT;
	nStateEmr			: INT;
	nState2				: INT;
	nState_IoT			: INT;
	bFaultFlag			: BOOL;
	nstateStop			: INT;
	fbTimerStop			: TON;
	timerStop			: ton;
	timerReset			: TON;
	nWriteData			: INT;
	TimerData			: TON;
	FbTimerModbus		: ARRAY [1..7] OF TON;
	fbEventlogger		: FB_Eventlogger;
	fbEventButton		: FB_EventButton;
	nstatechange		: INT;
	bWriteAlarm			: BOOL;
END_VAR

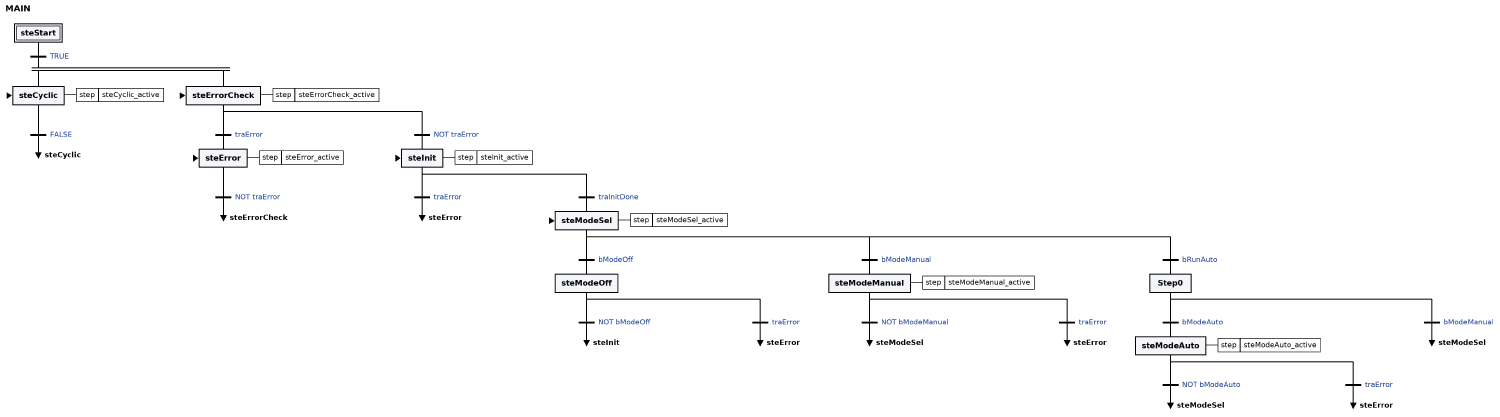
INITIAL_STEP steStart:
END_STEP
TRANSITION FROM steStart TO (steCyclic, steErrorCheck)
    := TRUE;
END_TRANSITION
STEP steCyclic:
    steCyclic_active(N);  // step action
END_STEP
TRANSITION FROM steCyclic TO steCyclic
    := FALSE;
END_TRANSITION
STEP steErrorCheck:
    steErrorCheck_active(N);  // step action
END_STEP
TRANSITION FROM steErrorCheck TO steError
    := traError;
END_TRANSITION
STEP steError:
    steError_active(N);  // step action
END_STEP
TRANSITION FROM steError TO steErrorCheck
    := NOT traError;
END_TRANSITION
TRANSITION FROM steErrorCheck TO steInit
    := NOT traError;
END_TRANSITION
STEP steInit:
    steInit_active(N);  // step action
END_STEP
TRANSITION FROM steInit TO steError
    := traError;
END_TRANSITION
TRANSITION FROM steInit TO steModeSel
    := traInitDone;
END_TRANSITION
STEP steModeSel:
    steModeSel_active(N);  // step action
END_STEP
TRANSITION FROM steModeSel TO steModeOff
    := bModeOff;
END_TRANSITION
STEP steModeOff:
END_STEP
TRANSITION FROM steModeOff TO steInit
    := NOT bModeOff;
END_TRANSITION
TRANSITION FROM steModeOff TO steError
    := traError;
END_TRANSITION
TRANSITION FROM steModeSel TO steModeManual
    := bModeManual;
END_TRANSITION
STEP steModeManual:
    steModeManual_active(N);  // step action
END_STEP
TRANSITION FROM steModeManual TO steModeSel
    := NOT bModeManual;
END_TRANSITION
TRANSITION FROM steModeManual TO steError
    := traError;
END_TRANSITION
TRANSITION FROM steModeSel TO Step0
    := bRunAuto;
END_TRANSITION
STEP Step0:
END_STEP
TRANSITION FROM Step0 TO steModeAuto
    := bModeAuto;
END_TRANSITION
TRANSITION FROM Step0 TO steModeSel
    := bModeManual;
END_TRANSITION
STEP steModeAuto:
    steModeAuto_active(N);  // step action
END_STEP
TRANSITION FROM steModeAuto TO steModeSel
    := NOT bModeAuto;
END_TRANSITION
TRANSITION FROM steModeAuto TO steError
    := traError;
END_TRANSITION

ACTION ListError:
Err_T(CLK := bError1);
Wrn_T(CLK := bWarning);

IF i > 100 THEN
	i := 100;
END_IF
		
CASE nState OF 
	0:
		IF Err_T.Q THEN
			nState := 1;
		ELSIF Wrn_T.Q THEN
			bWrn := TRUE;
			nState := 10;
		END_IF

	1:
		CASE nErrorID OF
			1:
				stErrorTxt := "E1_1.Lỗi hết hũ trạm 1 [kiểm tra U1I5-2]";
				stErrorTxt1 := 'E1_1.The jar is empty line 1 [check U1I5-2]';
				fbEventlogger(eventClass := TC_EVENTS.Entobel.Event1.uuidEventClass, nEventID := DINT_TO_UDINT(nErrorID));
			2:
				stErrorTxt := "E2_1.Lỗi hũ bị kẹt trạm 1 [kiểm tra U1I5-6]";
				stErrorTxt1 := 'E2_1.The jar  is trapped line 1 [check U1I5-6]';
				fbEventlogger(eventClass := TC_EVENTS.Entobel.Event2.uuidEventClass, nEventID := DINT_TO_UDINT(nErrorID));
			3:
				stErrorTxt := "E3_1.Lỗi ben chặn hũ trên rút về trạm 1 [kiểm tra U1I5-3]" ;
				stErrorTxt1 := 'E3_1.The upper cylinder retract  is faulty line 1 [check U1I5-3]';
				fbEventlogger(eventClass := TC_EVENTS.Entobel.Event3.uuidEventClass, nEventID := DINT_TO_UDINT(nErrorID));
			4:
				stErrorTxt := "E4_1.Lỗi ben chặn hũ dưới rút về trạm 1 [kiểm tra U1I5-4]";
				stErrorTxt1 := 'E4_1.The lower cylinder retract  is faulty line 1 [check U1I5-4]';
				fbEventlogger(eventClass := TC_EVENTS.Entobel.Event4.uuidEventClass, nEventID := DINT_TO_UDINT(nErrorID));
			5:
				stErrorTxt := "E5_1.Lỗi ben chặn hũ dưới đẩy ra trạm 1 [kiểmtra U1I5-5]";
				stErrorTxt1 := 'E5_1.The lower cylinder extend  is faulty line 1 [check U1I5-5]';
				fbEventlogger(eventClass := TC_EVENTS.Entobel.Event5.uuidEventClass, nEventID := DINT_TO_UDINT(nErrorID));
			6:
				stErrorTxt := "E6_1.Lỗi biến tần đảo thức ăn trạm 1 [kiểm tra biến tần 4]";
				stErrorTxt1 := 'E6_1.The inverter of agitator motor fault line 1 [check U1I5-6]';
				fbEventlogger(eventClass := TC_EVENTS.Entobel.Event6.uuidEventClass, nEventID := DINT_TO_UDINT(nErrorID));
			7:
				stErrorTxt := "E7_1.Lỗi driver chia thức ăn trạm 1 [kiểm tra driver 2]";
				stErrorTxt1 := 'E7_1.The driver of dispenser motor fault line 1 [check driver 2]';
				fbEventlogger(eventClass := TC_EVENTS.Entobel.Event7.uuidEventClass, nEventID := DINT_TO_UDINT(nErrorID));
			8:
				stErrorTxt := "E8_1.Lỗi ben chặn sâu rút về trạm 1 [kiểm tra U1I5-7]";
				stErrorTxt1 := 'E8_1.The cylinder blocking worm retract  is faulty line 1 [check U1I5-7]';
				fbEventlogger(eventClass := TC_EVENTS.Entobel.Event8.uuidEventClass, nEventID := DINT_TO_UDINT(nErrorID));
			9:
				stErrorTxt := "E9_1.Lỗi biến tần phểu rung sâu trạm 1 [kiểm tra biến tần 5]";
				stErrorTxt1 := 'E9_1.The inverter of vibrating funnel fault line 1 [check inverter 5]';
				fbEventlogger(eventClass := TC_EVENTS.Entobel.Event9.uuidEventClass, nEventID := DINT_TO_UDINT(nErrorID));
			10:
				stErrorTxt := "E10_1.Lỗi hết nắp trạm 1 [kiểm tra U1I5-8]";
				stErrorTxt1 := 'E10_1.The lid is empty line 1 [check U1I5-8]';
				fbEventlogger(eventClass := TC_EVENTS.Entobel.Event10.uuidEventClass, nEventID := DINT_TO_UDINT(nErrorID));
			11:
				stErrorTxt := "E11_1.Lỗi ben chặn nắp rút về trạm 1 [kiểm tra U1I6-1]";
				stErrorTxt1 := 'E11_1.The cylinder blocking the lid retract is faulty line 1 [check U1I6-1]';
				fbEventlogger(eventClass := TC_EVENTS.Entobel.Event11.uuidEventClass, nEventID := DINT_TO_UDINT(nErrorID));
			12:
				stErrorTxt := "E12-1.Lỗi ben chặn nắp đẩy ra trạm 1 [kiểm tra U1I6-2]";
				stErrorTxt1 := 'E12_1.The cylinder blocking the lid extend is faulty line 1 [check U1I6-2]';
				fbEventlogger(eventClass := TC_EVENTS.Entobel.Event12.uuidEventClass, nEventID := DINT_TO_UDINT(nErrorID));
			13:
				stErrorTxt := "E13_1.Lỗi ben hút/thả nắp rút về trạm 1 [kiểm tra U1I6-3]";
				stErrorTxt1 := 'E13_1.The cylinder sucking the lid retract is faulty line 1 [check U1I6-3]';
				fbEventlogger(eventClass := TC_EVENTS.Entobel.Event13.uuidEventClass, nEventID := DINT_TO_UDINT(nErrorID));
			14:
				stErrorTxt := "E14_1.Lỗi ben hút/thả nắp đẩy ra trạm 1 [kiểm tra U1I6-4]";
				stErrorTxt1 := 'E14_1.The cylinder sucking the lid extend is faulty line 1 [check U1I6-4]';
				fbEventlogger(eventClass := TC_EVENTS.Entobel.Event14.uuidEventClass, nEventID := DINT_TO_UDINT(nErrorID));
			15:
				stErrorTxt := "E15_1.Lỗi ben dập nắp rút về trạm 1 [kiểm tra U1I6-6]";
				stErrorTxt1 := 'E15_1.The cylinder pressing the lid retract is faulty line 1 [check U1I6-6]';
				fbEventlogger(eventClass := TC_EVENTS.Entobel.Event15.uuidEventClass, nEventID := DINT_TO_UDINT(nErrorID));
			16:
				stErrorTxt := "E16_1.Lỗi ben dập nắp đẩy ra trạm 1 [kiểm tra U1I6-7]";
				stErrorTxt1 := 'E16_1.The cylinder pressing the lid extend is faulty line 1 [check U1I6-7]';
				fbEventlogger(eventClass := TC_EVENTS.Entobel.Event16.uuidEventClass, nEventID := DINT_TO_UDINT(nErrorID));
			17:
				stErrorTxt := "E17_1.Lỗi ben lượt ra/vào rút về trạm 1 [kiểm tra U1I6-8]";
				stErrorTxt1 := 'E17_1.The comb cylinder retract is faulty line 1 [check U1I6-8]';
				fbEventlogger(eventClass := TC_EVENTS.Entobel.Event17.uuidEventClass, nEventID := DINT_TO_UDINT(nErrorID));
			18:
				stErrorTxt := "E18_1.Lỗi ben lượt ra/vào đẩy ra trạm 1 [kiểm tra U1I7-1]";
				stErrorTxt1 := 'E18_1.The comb cylinder extend is faulty line 1 [check U1I7-1]';
				fbEventlogger(eventClass := TC_EVENTS.Entobel.Event18.uuidEventClass, nEventID := DINT_TO_UDINT(nErrorID));
			19:
				stErrorTxt := "E19_1.Lỗi ben kẹp hũ rút về trạm 1 [kiểm tra U1I7-4]";
				stErrorTxt1 := 'E19_1.The clap cylinder retract is faulty line 1 [check U1I7-4]';
				fbEventlogger(eventClass := TC_EVENTS.Entobel.Event19.uuidEventClass, nEventID := DINT_TO_UDINT(nErrorID));
			20:
				stErrorTxt := "E20_1.Lỗi ben kẹp hũ đẩy ra trạm 1 [kiểm tra U1I7-5]";	
				stErrorTxt1 := 'E20_1.The clap cylinder extend is faulty line 1 [check U1I7-5]';
				fbEventlogger(eventClass := TC_EVENTS.Entobel.Event20.uuidEventClass, nEventID := DINT_TO_UDINT(nErrorID));
			21:
				stErrorTxt := "E21_1.Lỗi ben di chuyển lượt rút về trạm 1 [kiểm tra U1I7-2]";	
				stErrorTxt1 := 'E21_1.The cylinder moving comb retract is faulty line 1 [check U1I7-2]';
				fbEventlogger(eventClass := TC_EVENTS.Entobel.Event21.uuidEventClass, nEventID := DINT_TO_UDINT(nErrorID));
			22:
				stErrorTxt := "E22_1.Lỗi ben di chuyển lượt đẩy ra trạm 1 [kiểm tra U1I7-3]";
				stErrorTxt1 := 'E22_1.The cylinder moving comb extend is faulty line 1 [check U1I7-3]';
				fbEventlogger(eventClass := TC_EVENTS.Entobel.Event22.uuidEventClass, nEventID := DINT_TO_UDINT(nErrorID));
			45:
				stErrorTxt := "E23_1.Lỗi mất hũ khi đang cân thức ăn trạm 1 [kiểm tra U1I7-6]";
				stErrorTxt1 := 'E23_1.The jar is missed when weighting food line 1 [check U1I7-6]';
				fbEventlogger(eventClass := TC_EVENTS.Entobel.Event45.uuidEventClass, nEventID := DINT_TO_UDINT(nErrorID));
			47:
				stErrorTxt := "E24_1.Lỗi mất hũ khi đang cân sâu trạm 1 [kiểm tra U1I7-7]";
				stErrorTxt1 := 'E24_1.The jar is missed when weighting larvae line 1 [check U1I7-7]';
				fbEventlogger(eventClass := TC_EVENTS.Entobel.Event47.uuidEventClass, nEventID := DINT_TO_UDINT(nErrorID));
			49:
				stErrorTxt := "E25_1.Lỗi hút không được nắp trạm 1 [kiểm tra U1I6-5]";
				stErrorTxt1 := 'E25_1.Failed to suction the lid line 1 [check U1I6-5]';
				fbEventlogger(eventClass := TC_EVENTS.Entobel.Event49.uuidEventClass, nEventID := DINT_TO_UDINT(nErrorID));
			51:
				stErrorTxt := "E26_1.Lỗi nắp đã được hút trạm 1 [kiểm tra U1I6-5]";
				stErrorTxt1 := 'E26_1.The lid is still on the valve line 1 [check U1I5-6]';	
				fbEventlogger(eventClass := TC_EVENTS.Entobel.Event51.uuidEventClass, nEventID := DINT_TO_UDINT(nErrorID));
			53:
				stErrorTxt := "E27_1.Lỗi an toàn cửa 1 [kiểm tra U1I7-8]";	
				stErrorTxt1 := 'E27_1.The safety door 1 is error [check U1I7-8]';	
				fbEventlogger(eventClass := TC_EVENTS.Entobel.Event53.uuidEventClass, nEventID := DINT_TO_UDINT(nErrorID));
			54:
				stErrorTxt := "E28_1.Lỗi an toàn cửa 2 [kiểm tra U1I7-9]";
				stErrorTxt1 := 'E28_1.The safety door 2 is error [check U1I7-9]';	
				fbEventlogger(eventClass := TC_EVENTS.Entobel.Event54.uuidEventClass, nEventID := DINT_TO_UDINT(nErrorID));
			55:
				stErrorTxt := "E29_1.Lỗi an toàn cửa 3 [kiểm tra U1I7-10]";
				stErrorTxt1 := 'E29_1.The safety door 3 is error [check U1I7-10]';
				fbEventlogger(eventClass := TC_EVENTS.Entobel.Event55.uuidEventClass, nEventID := DINT_TO_UDINT(nErrorID));	
			56: 
				stErrorTxt := "E30_1.Lỗi quá cân thức ăn trạm 1 [kiểm tra cân thức ăn]";
				stErrorTxt1 := 'E30_1.Overload weightfood [check U1I5-6]';	
				fbEventlogger(eventClass := TC_EVENTS.Entobel.Event56.uuidEventClass, nEventID := DINT_TO_UDINT(nErrorID));
			57: 
				stErrorTxt := "E31_1.Lỗi quá cân sâu trạm 1 [kiểm tra cân sâu]";
				stErrorTxt1 := 'E30_1.Overload weightLarvae [check U1I5-6]';
				fbEventlogger(eventClass := TC_EVENTS.Entobel.Event57.uuidEventClass, nEventID := DINT_TO_UDINT(nErrorID));	
			60:
				stErrorTxt := "E32_1.Lỗi ben hút/thả hũ đẩy ra trạm 1 [kiểm tra U1I7-11]";
				stErrorTxt1 := 'E32_1.The cylinder sucking the jar is faulty line 1 [check U1I7-11]';
				fbEventlogger(eventClass := TC_EVENTS.Entobel.Event60.uuidEventClass, nEventID := DINT_TO_UDINT(nErrorID)); 
			64:
				stErrorTxt := "E33_1.Lỗi Modbus thiết bị 3";
				stErrorTxt1 := 'E33_1.Error Modbus device 3';
				fbEventlogger(eventClass := TC_EVENTS.Entobel.Event64.uuidEventClass, nEventID := DINT_TO_UDINT(nErrorID));	
			65:
				stErrorTxt := "E34_1.Lỗi Modbus thiết bị 4";
				stErrorTxt1 := 'E34_1.Error Modbus device 4';
				fbEventlogger(eventClass := TC_EVENTS.Entobel.Event65.uuidEventClass, nEventID := DINT_TO_UDINT(nErrorID));	
			66:
				stErrorTxt := "E35_1.Lỗi Modbus thiết bị 5";
				stErrorTxt1 := 'E35_1.Error Modbus device 5';
				fbEventlogger(eventClass := TC_EVENTS.Entobel.Event66.uuidEventClass, nEventID := DINT_TO_UDINT(nErrorID));	
			68:
				stErrorTxt := "E36_1.Lỗi Modbus thiết bị 7";
				stErrorTxt1 := 'E36_1.Error Modbus device 7';
				fbEventlogger(eventClass := TC_EVENTS.Entobel.Event68.uuidEventClass, nEventID := DINT_TO_UDINT(nErrorID));	
			69:
				stErrorTxt := "E37_1.Lỗi đầu cân thức ăn Mettler Toledo 1";
				stErrorTxt1 := 'E37_1.Error Mettler Toledo 1';
				fbEventlogger(eventClass := TC_EVENTS.Entobel.Event69.uuidEventClass, nEventID := DINT_TO_UDINT(nErrorID));	
			70:
				stErrorTxt := "E38_1.Lỗi đầu cân sâu Mettler Toledo 2";
				stErrorTxt1 := 'E38_1.Error Mettler Toledo 2';
				fbEventlogger(eventClass := TC_EVENTS.Entobel.Event70.uuidEventClass, nEventID := DINT_TO_UDINT(nErrorID));	
			73:
				stErrorTxt := "E39_1.Lỗi ben chặn sâu đẩy ra trạm 1 [kiểm tra U1I5-7]";
				stErrorTxt1 := 'E39_1.The cylinder blocking worm extend  is faulty line 1';
				fbEventlogger(eventClass := TC_EVENTS.Entobel.Event73.uuidEventClass, nEventID := DINT_TO_UDINT(nErrorID));	
			75:
				stErrorTxt := "E40_1.Lỗi thiếu khí đầu vào [kiểm tra U1I7-13]";
				stErrorTxt1 := 'E40_1.Error of lack of input air [check U1I7-13]';
				fbEventlogger(eventClass := TC_EVENTS.Entobel.Event75.uuidEventClass, nEventID := DINT_TO_UDINT(nErrorID));	
			76:
				stErrorTxt := "E41_1.Lỗi hết thức ăn trạm 1";
				stErrorTxt1 := 'E41_1.Error running out of food line 1';
				fbEventlogger(eventClass := TC_EVENTS.Entobel.Event76.uuidEventClass, nEventID := DINT_TO_UDINT(nErrorID));	
			77:
				stErrorTxt := "E42_1.Lỗi hết sâu trạm 1";
				stErrorTxt1 := 'E42_1.Error running out of larvae line 1';
				fbEventlogger(eventClass := TC_EVENTS.Entobel.Event78.uuidEventClass, nEventID := DINT_TO_UDINT(nErrorID));		
			98:
				stErrorTxt := "E98_1.Dừng khẩn [kiểm tra Emergency]";
				stErrorTxt1 := 'E98_1.Emergency Stop [check Emergency]';
				fbEventlogger(eventClass := TC_EVENTS.Entobel.Event98.uuidEventClass, nEventID := DINT_TO_UDINT(nErrorID));	 
			99: 
				stErrorTxt := "E99_1.Lỗi biến tần băng tải đầu ra [kiểm tra biến tần 3]";
				stErrorTxt1 := 'E99_1.The inverter of conveyor out [check inverter 3]';	
				fbEventlogger(eventClass := TC_EVENTS.Entobel.Event99.uuidEventClass, nEventID := DINT_TO_UDINT(nErrorID));
		END_CASE
		IF i <> 1 THEN
			FOR	k := i TO 2 BY -1 DO
				nErrorIDList1[k].nErrorID 	 := nErrorIDList1[k-1].nErrorID;
				nErrorIDList1[k].ErrorTime   := nErrorIDList1[k-1].ErrorTime;
				nErrorIDList1[k].ErrorStatus := nErrorIDList1[k-1].ErrorStatus;	
			END_FOR		
		END_IF 
		nErrorIDList1[1].nErrorID := nErrorID;
		nErrorIDList1[1].ErrorTime := SYSTEMTIME_TO_DT(GetLocalSystemTime.systemTime);
		nErrorIDList1[1].ErrorStatus := 1;
		nStatus1	:= 'ERROR';
		i := i + 1;
		bWarning := FALSE;
		bTo_alarm_side := TRUE;
		nState := 2;
	2:
		bWriteAlarm	:= TRUE;
		bSirens := TRUE;
		nState := 3;
	3:
		IF NOT bError1 THEN
			nState 	:= 0;
			bSirens := FALSE;
		END_IF
	10:
		CASE nWarningID OF
			101:
				stWarningTxt := "W1_1.Cảnh báo hết hũ trạm 1[kiểm tra U1I5-2]";
				stWarningTxt1 := 'W1_1.Warning out of jar line 1 [check U1I5-2]';
				fbEventlogger(eventClass := TC_EVENTS.Entobel.Event101.uuidEventClass, nEventID := DINT_TO_UDINT(nWarningID));
			102:
				stWarningTxt := "W2_1.Cảnh báo hết nắp trạm 1[kiểm tra U1I5-8]";
				stWarningTxt1 := 'W2_1.Warning out of lid line 1 [check U1I5-8]';
				fbEventlogger(eventClass := TC_EVENTS.Entobel.Event102.uuidEventClass, nEventID := DINT_TO_UDINT(nWarningID));
			103:
				stWarningTxt := "W3_1.Cảnh báo hết thức ăn trạm 1";
				stWarningTxt1 := 'W3_1.Warning running out of food line 1';
				fbEventlogger(eventClass := TC_EVENTS.Entobel.Event103.uuidEventClass, nEventID := DINT_TO_UDINT(nWarningID));
			104:
				stWarningTxt := "W4_1.Cảnh báo cân quá khối lượng thức ăn trạm 1";
				stWarningTxt1 := 'W4_1.Warning food weight exceeds limit line 1';
				fbEventlogger(eventClass := TC_EVENTS.Entobel.Event104.uuidEventClass, nEventID := DINT_TO_UDINT(nWarningID));
			105:
				stWarningTxt := "W5_1.Cảnh báo hết sâu trạm 1";
				stWarningTxt1 := 'W5_1.Warning running out of larvae line 1';
				fbEventlogger(eventClass := TC_EVENTS.Entobel.Event105.uuidEventClass, nEventID := DINT_TO_UDINT(nWarningID));
			106:
				stWarningTxt := "W6_1.Canh bao can qua khoi luong sau tram 1";
				stWarningTxt1 := 'W6_1.Warning larvae weight exceeds limit line 1';
				fbEventlogger(eventClass := TC_EVENTS.Entobel.Event106.uuidEventClass, nEventID := DINT_TO_UDINT(nWarningID));
			107:
				stWarningTxt := "W7_1.Cảnh báo dập nắp không vô trạm 1[kiểm tra U1I6-7]";
				stWarningTxt1 := 'W7_1.Warning do not press lid inward line 1 [check U1I6-7]';
				fbEventlogger(eventClass := TC_EVENTS.Entobel.Event107.uuidEventClass, nEventID := DINT_TO_UDINT(nWarningID));
			115:
				stWarningTxt := "W8_1.Cảnh báo mất kết nối với PC Advantech [kiểm tra PC]";
				stWarningTxt1 := 'W8_1.Warning disconnect to PC Advantech [check PC]';	
				bAlarm_Iot := TRUE;	
		END_CASE
		IF i <> 1 THEN
			FOR	k := i TO 2 BY -1 DO
				nErrorIDList1[k].nErrorID 	 := nErrorIDList1[k-1].nErrorID;
				nErrorIDList1[k].ErrorTime   := nErrorIDList1[k-1].ErrorTime;
				nErrorIDList1[k].ErrorStatus := nErrorIDList1[k-1].ErrorStatus;		
			END_FOR		
		END_IF 
		nErrorIDList1[1].nErrorID := nWarningID;
		nErrorIDList1[1].ErrorTime := SYSTEMTIME_TO_DT(GetLocalSystemTime.systemTime);
		nErrorIDList1[1].ErrorStatus := 1;
		nStatus1	:= 'WARNING';
		i := i + 1;
		nState := 11;
	11:
		bWriteAlarm	:= TRUE;
		bSirens := TRUE;
		nState := 12;
	12:
		bWarning := FALSE;
		nState := 0;		
END_CASE

IF bclearall THEN
	FOR k := 1 TO 100 DO
		AlarmList[1,k] := "";
		AlarmList[2,k] := "";	
		AlarmList[3,k] := "";
		AlarmList[4,k] := "";	
		AlarmList3[1,k] := '';
		AlarmList3[2,k] := '';	
		AlarmList3[3,k] := '';
		AlarmList3[4,k] := '';	
	END_FOR
	i := 1;
END_IF

IF username <> '' THEN
	IF getuser = 'Operator' THEN
		IF NOT bSafetyDoor1 THEN
			F_SetError(53,nLine := 3);
		ELSIF NOT bSafetyDoor2 THEN
			F_SetError(54,nLine := 3);	
		ELSIF NOT bSafetyDoor3 THEN
			F_SetError(55,nLine := 3);	
		END_IF
		bypass := FALSE;
		hienthibypass := FALSE;
	ELSIF getuser = 'Engineer' THEN
		hienthibypass := TRUE;
		IF NOT bypass THEN
			IF NOT bSafetyDoor1 THEN
				F_SetError(53,nLine := 3);
			ELSIF NOT bSafetyDoor2 THEN
				F_SetError(54,nLine := 3);	
			ELSIF NOT bSafetyDoor3 THEN
				F_SetError(55,nLine := 3);	
			END_IF
		END_IF
	END_IF
END_IF
IF username <> '' THEN
	IF Error[1] THEN 
		(*IF ErrorID[1] = 150 OR ErrorID[1] = 32 THEN
			FbTimerModbus[1](IN := FALSE, PT := T#1S);
		ELSE*)
			//FbTimerModbus[1](IN := TRUE, PT := T#1S);
			//IF FbTimerModbus[1].Q  THEN
				F_SetError(62,nLine := 2);
			//END_IF
		//END_IF
	ELSE
		FbTimerModbus[1](IN := FALSE);
	END_IF
	
	IF Error[2] THEN
		(*IF ErrorID[2] = 150 OR ErrorID[2] = 32 THEN
			FbTimerModbus[2](IN := FALSE, PT := T#1S);
		ELSE*)
			//FbTimerModbus[2](IN := TRUE, PT := T#1S);
			//IF FbTimerModbus[2].Q THEN
				F_SetError(63,nLine := 2);
			//END_IF
		//END_IF
	ELSE
		FbTimerModbus[2](IN := FALSE);
	END_IF
	
	IF Error[3] THEN
		(*IF ErrorID[3] = 150 OR ErrorID[3] = 32 THEN
			FbTimerModbus[3](IN := FALSE, PT := T#1S);
		ELSE*)
			//FbTimerModbus[3](IN := TRUE, PT := T#1S);
			//IF FbTimerModbus[3].Q THEN
				F_SetError(64,nLine := 3);
				PR_Conveyor_Out.Stop();
				bRun := FALSE;
			//END_IF
		//END_IF
	ELSE
		FbTimerModbus[3](IN := FALSE);
	END_IF
	
	IF Error[4] THEN
		(*IF ErrorID[4] = 150 OR ErrorID[4] = 32 THEN
			FbTimerModbus[4](IN := FALSE, PT := T#1S);
		ELSE *)
			//FbTimerModbus[4](IN := TRUE, PT := T#1S);
			//IF FbTimerModbus[4].Q THEN
				F_SetError(65,nLine := 1);
			//END_IF
		//END_IF
	ELSE
		FbTimerModbus[4](IN := FALSE);
	END_IF
	
	IF Error[5] THEN
		(*IF ErrorID[5] = 150 OR ErrorID[5] = 32 THEN
			FbTimerModbus[5](IN := FALSE, PT := T#1S);
		ELSE*)
			//FbTimerModbus[5](IN := TRUE, PT := T#1S);
			//IF FbTimerModbus[5].Q THEN
				F_SetError(66,nLine := 1);
			//END_IF
		//END_IF
	ELSE
		FbTimerModbus[5](IN := FALSE);
	END_IF
	
	IF Error[6] THEN
		(*IF ErrorID[6] = 150 OR ErrorID[6] = 32 THEN
			FbTimerModbus[6](IN := FALSE, PT := T#1S);
		ELSE*)
			//FbTimerModbus[6](IN := TRUE, PT := T#1S);
			//IF FbTimerModbus[6].Q THEN
				F_SetError(67,nLine := 2);
			//END_IF
		//END_IF
	ELSE
		FbTimerModbus[6](IN := FALSE);
	END_IF
	
	IF Error[7] THEN
		(*IF ErrorID[2] = 150 OR ErrorID[7] = 32 THEN
			FbTimerModbus[7](IN := FALSE, PT := T#1S);
		ELSE*)
			//FbTimerModbus[7](IN := TRUE, PT := T#1S);
			//IF FbTimerModbus[7].Q THEN
				F_SetError(68,nLine := 1);
			//END_IF
		//END_IF
	ELSE
		FbTimerModbus[7](IN := FALSE);
	END_IF
END_IF

IF username <> '' THEN
	IF bCheckVan THEN
		F_SetError(75,nLine := 3);
	END_IF
END_IF

IF bError1 AND bError2 AND (nErrorId = 99 OR nErrorID = 64) THEN
	PR_Conveyor_Out.Stop();
END_IF 

IF bWrn THEN
	bWrn2 := FALSE;
ELSIF bWrn2 THEN
	bWrn := FALSE;
END_IF

IF bWrn OR bWrn2 THEN
	bxoa := TRUE;
ELSE 
	bxoa := FALSE;
END_IF

CASE nStateEmr OF 
	0:
		IF NOT bEmer THEN
			F_SetError(98,nLine := 3);
			nStateEmr := 1;
		END_IF
	1:
		IF bEmer THEN
			nStateEmr := 0;
		END_IF
END_CASE
END_ACTION

ACTION MapRtig:
IF getuser = 'Operator' THEN
	CASE nstatechange OF 
		0:
			//line 1
			fFast_Speed_line1_change						:= PR_Line01.fFast_Speed;//FoodWeight
			fSlow_Speed_1_line1_change						:= PR_Line01.fSlow_Speed_1;
			fSlow_Speed_2_line1_change						:= PR_Line01.fSlow_Speed_2;
			fDerisedWeight_Food_line1_change				:= PR_Line01.fDerisedWeight_Food;
			fChangeMode_Food_1_line1_change					:= PR_Line01.fChangeMode_Food_1;
			fChangeMode_Food_2_line1_change					:= PR_Line01.fChangeMode_Food_2;
			fPerStop_Food_line1_change						:= PR_Line01.fPerStop_Food;
			fTimer_Check_Food_line1_change					:= PR_Line01.fTimer_Check_Food;
			fDelta_Food_line1_change						:= PR_Line01.fDelta_Food;
			fFast_Speed_vibrating_funnel_line1_change		:= PR_Line01.fFast_Speed_vibrating_funnel;//WormWeight
			fSlow_Speed_vibrating_funnel_1_line1_change		:= PR_Line01.fSlow_Speed_vibrating_funnel_1;
			fSlow_Speed_vibrating_funnel_2_line1_change		:= PR_Line01.fSlow_Speed_vibrating_funnel_2;
			fDerisedWeight_Worm_line1_change				:= PR_Line01.fDerisedWeight_Worm;
			fChangeMode_Worm_1_line1_change					:= PR_Line01.fChangeMode_Worm_1;
			fChangeMode_Worm_2_line1_change					:= PR_Line01.fChangeMode_Worm_2;
			fPerStop_Worm_line1_change						:= PR_Line01.fPerStop_Worm;
			fTimer_Check_Worm_line1_change					:= PR_Line01.fTimer_Check_Worm;
			fDelta_Worm_line1_change						:= PR_Line01.fDelta_Worm;
			//line 2
			fFast_Speed_line2_change						:= PR_Line02.fFast_Speed;//FoodWeight
			fSlow_Speed_1_line2_change						:= PR_Line02.fSlow_Speed_1;
			fSlow_Speed_2_line2_change						:= PR_Line02.fSlow_Speed_2;
			fDerisedWeight_Food_line2_change				:= PR_Line02.fDerisedWeight_Food;
			fChangeMode_Food_1_line2_change					:= PR_Line02.fChangeMode_Food_1;
			fChangeMode_Food_2_line2_change					:= PR_Line02.fChangeMode_Food_2;
			fPerStop_Food_line2_change						:= PR_Line02.fPerStop_Food;
			fTimer_Check_Food_line2_change					:= PR_Line02.fTimer_Check_Food;
			fDelta_Food_line2_change						:= PR_Line02.fDelta_Food;
			fFast_Speed_vibrating_funnel_line2_change		:= PR_Line02.fFast_Speed_vibrating_funnel;//WormWeight
			fSlow_Speed_vibrating_funnel_1_line2_change		:= PR_Line02.fSlow_Speed_vibrating_funnel_1;
			fSlow_Speed_vibrating_funnel_2_line2_change		:= PR_Line02.fSlow_Speed_vibrating_funnel_2;
			fDerisedWeight_Worm_line2_change				:= PR_Line02.fDerisedWeight_Worm;
			fChangeMode_Worm_1_line2_change					:= PR_Line02.fChangeMode_Worm_1;
			fChangeMode_Worm_2_line2_change					:= PR_Line02.fChangeMode_Worm_2;
			fPerStop_Worm_line2_change						:= PR_Line02.fPerStop_Worm;
			fTimer_Check_Worm_line2_change					:= PR_Line02.fTimer_Check_Worm;
			fDelta_Worm_line2_change						:= PR_Line02.fDelta_Worm;
			nstatechange := 1;
		1:
			IF 	fFast_Speed_line1_change <> PR_Line01.fFast_Speed THEN
				fbEventButton(eventClass := TC_EVENTS.Entobel.Event150.uuidEventClass, nEventID := 150,
							  sString := REAL_TO_STRING(PR_Line01.fFast_Speed));
				nstatechange := 0;
			ELSIF fSlow_Speed_1_line1_change <> PR_Line01.fSlow_Speed_1 THEN
				fbEventButton(eventClass := TC_EVENTS.Entobel.Event151.uuidEventClass, nEventID := 151,
							  sString := REAL_TO_STRING(PR_Line01.fSlow_Speed_1)); 
				nstatechange := 0;
			ELSIF fSlow_Speed_2_line1_change <> PR_Line01.fSlow_Speed_2 THEN
				fbEventButton(eventClass := TC_EVENTS.Entobel.Event152.uuidEventClass, nEventID := 152,
							  sString := REAL_TO_STRING(PR_Line01.fSlow_Speed_2)); 
				nstatechange := 0;
			ELSIF fDerisedWeight_Food_line1_change <> PR_Line01.fDerisedWeight_Food THEN
				fbEventButton(eventClass := TC_EVENTS.Entobel.Event153.uuidEventClass, nEventID := 153,
							  sString := REAL_TO_STRING(PR_Line01.fDerisedWeight_Food)); 
				nstatechange := 0;
			ELSIF fChangeMode_Food_1_line1_change <> PR_Line01.fChangeMode_Food_1 THEN
				fbEventButton(eventClass := TC_EVENTS.Entobel.Event154.uuidEventClass, nEventID := 154,
							  sString := REAL_TO_STRING(PR_Line01.fChangeMode_Food_1)); 
				nstatechange := 0;
			ELSIF fChangeMode_Food_2_line1_change <> PR_Line01.fChangeMode_Food_2 THEN
				fbEventButton(eventClass := TC_EVENTS.Entobel.Event155.uuidEventClass, nEventID := 155,
							  sString := REAL_TO_STRING(PR_Line01.fChangeMode_Food_2)); 
				nstatechange := 0;
			ELSIF fPerStop_Food_line1_change <> PR_Line01.fPerStop_Food THEN
				fbEventButton(eventClass := TC_EVENTS.Entobel.Event156.uuidEventClass, nEventID := 156,
							  sString := REAL_TO_STRING(PR_Line01.fPerStop_Food)); 
				nstatechange := 0;
			ELSIF fTimer_Check_Food_line1_change <> PR_Line01.fTimer_Check_Food THEN
				fbEventButton(eventClass := TC_EVENTS.Entobel.Event157.uuidEventClass, nEventID := 157,
							  sString := REAL_TO_STRING(PR_Line01.fTimer_Check_Food)); 
				nstatechange := 0;
			ELSIF fDelta_Food_line1_change <> PR_Line01.fDelta_Food THEN
				fbEventButton(eventClass := TC_EVENTS.Entobel.Event158.uuidEventClass, nEventID := 158,
							  sString := REAL_TO_STRING(PR_Line01.fDelta_Food)); 
				nstatechange := 0;
			ELSIF fFast_Speed_vibrating_funnel_line1_change <> PR_Line01.fFast_Speed_vibrating_funnel THEN
					fbEventButton(eventClass := TC_EVENTS.Entobel.Event159.uuidEventClass, nEventID := 159,
							  sString := REAL_TO_STRING(PR_Line01.fFast_Speed_vibrating_funnel)); 
				nstatechange := 0;
			ELSIF fSlow_Speed_vibrating_funnel_1_line1_change <> PR_Line01.fSlow_Speed_vibrating_funnel_1 THEN
				fbEventButton(eventClass := TC_EVENTS.Entobel.Event160.uuidEventClass, nEventID := 160,
							  sString := REAL_TO_STRING(PR_Line01.fSlow_Speed_vibrating_funnel_1)); 
				nstatechange := 0;
			ELSIF fSlow_Speed_vibrating_funnel_2_line1_change <> PR_Line01.fSlow_Speed_vibrating_funnel_2 THEN
				fbEventButton(eventClass := TC_EVENTS.Entobel.Event161.uuidEventClass, nEventID := 161,
							  sString := REAL_TO_STRING(PR_Line01.fSlow_Speed_vibrating_funnel_2)); 
				nstatechange := 0;
			ELSIF fDerisedWeight_Worm_line1_change <> PR_Line01.fDerisedWeight_Worm THEN
				fbEventButton(eventClass := TC_EVENTS.Entobel.Event162.uuidEventClass, nEventID := 162,
							  sString := REAL_TO_STRING(PR_Line01.fDerisedWeight_Worm)); 
				nstatechange := 0;
			ELSIF fChangeMode_Worm_1_line1_change <> PR_Line01.fChangeMode_Worm_1 THEN
				fbEventButton(eventClass := TC_EVENTS.Entobel.Event163.uuidEventClass, nEventID := 163,
							  sString := REAL_TO_STRING(PR_Line01.fChangeMode_Worm_1)); 
				nstatechange := 0;
			ELSIF fChangeMode_Worm_2_line1_change <> PR_Line01.fChangeMode_Worm_2 THEN
				fbEventButton(eventClass := TC_EVENTS.Entobel.Event164.uuidEventClass, nEventID := 164,
							  sString := REAL_TO_STRING(PR_Line01.fChangeMode_Worm_2)); 
				nstatechange := 0;
			ELSIF fPerStop_Worm_line1_change <> PR_Line01.fPerStop_Worm THEN
				fbEventButton(eventClass := TC_EVENTS.Entobel.Event165.uuidEventClass, nEventID := 165,
							  sString := REAL_TO_STRING(PR_Line01.fPerStop_Worm)); 
				nstatechange := 0;
			ELSIF fTimer_Check_Worm_line1_change <> PR_Line01.fTimer_Check_Worm THEN
				fbEventButton(eventClass := TC_EVENTS.Entobel.Event166.uuidEventClass, nEventID := 166,
							  sString := REAL_TO_STRING(PR_Line01.fTimer_Check_Worm)); 
				nstatechange := 0;
			ELSIF fDelta_Worm_line1_change <> PR_Line01.fDelta_Worm THEN
				fbEventButton(eventClass := TC_EVENTS.Entobel.Event167.uuidEventClass, nEventID := 167,
							  sString := REAL_TO_STRING(PR_Line01.fDelta_Worm)); 
				nstatechange := 0;
			ELSIF 	fFast_Speed_line2_change <> PR_Line02.fFast_Speed THEN
				fbEventButton(eventClass := TC_EVENTS.Entobel.Event168.uuidEventClass, nEventID := 168,
							  sString := REAL_TO_STRING(PR_Line02.fFast_Speed));
				nstatechange := 0;
			ELSIF fSlow_Speed_1_line2_change <> PR_Line02.fSlow_Speed_1 THEN
				fbEventButton(eventClass := TC_EVENTS.Entobel.Event169.uuidEventClass, nEventID := 169,
							  sString := REAL_TO_STRING(PR_Line02.fSlow_Speed_1)); 
				nstatechange := 0;
			ELSIF fSlow_Speed_2_line2_change <> PR_Line02.fSlow_Speed_2 THEN
				fbEventButton(eventClass := TC_EVENTS.Entobel.Event170.uuidEventClass, nEventID := 170,
							  sString := REAL_TO_STRING(PR_Line02.fSlow_Speed_2)); 
				nstatechange := 0;
			ELSIF fDerisedWeight_Food_line2_change <> PR_Line02.fDerisedWeight_Food THEN
				fbEventButton(eventClass := TC_EVENTS.Entobel.Event171.uuidEventClass, nEventID := 171,
							  sString := REAL_TO_STRING(PR_Line02.fDerisedWeight_Food)); 
				nstatechange := 0;
			ELSIF fChangeMode_Food_1_line2_change <> PR_Line02.fChangeMode_Food_1 THEN
				fbEventButton(eventClass := TC_EVENTS.Entobel.Event172.uuidEventClass, nEventID := 172,
							  sString := REAL_TO_STRING(PR_Line02.fChangeMode_Food_1)); 
				nstatechange := 0;
			ELSIF fChangeMode_Food_2_line2_change <> PR_Line02.fChangeMode_Food_2 THEN
				fbEventButton(eventClass := TC_EVENTS.Entobel.Event173.uuidEventClass, nEventID := 173,
							  sString := REAL_TO_STRING(PR_Line02.fChangeMode_Food_2)); 
				nstatechange := 0;
			ELSIF fPerStop_Food_line2_change <> PR_Line02.fPerStop_Food THEN
				fbEventButton(eventClass := TC_EVENTS.Entobel.Event174.uuidEventClass, nEventID := 174,
							  sString := REAL_TO_STRING(PR_Line02.fPerStop_Food)); 
				nstatechange := 0;
			ELSIF fTimer_Check_Food_line2_change <> PR_Line02.fTimer_Check_Food THEN
				fbEventButton(eventClass := TC_EVENTS.Entobel.Event175.uuidEventClass, nEventID := 175,
							  sString := REAL_TO_STRING(PR_Line02.fTimer_Check_Food)); 
				nstatechange := 0;
			ELSIF fDelta_Food_line2_change <> PR_Line02.fDelta_Food THEN
				fbEventButton(eventClass := TC_EVENTS.Entobel.Event176.uuidEventClass, nEventID := 176,
							  sString := REAL_TO_STRING(PR_Line02.fDelta_Food)); 
				nstatechange := 0;
			ELSIF fFast_Speed_vibrating_funnel_line2_change <> PR_Line02.fFast_Speed_vibrating_funnel THEN
				fbEventButton(eventClass := TC_EVENTS.Entobel.Event185.uuidEventClass, nEventID := 185,
							  sString := REAL_TO_STRING(PR_Line02.fFast_Speed_vibrating_funnel)); 
				nstatechange := 0;
			ELSIF fSlow_Speed_vibrating_funnel_1_line2_change <> PR_Line02.fSlow_Speed_vibrating_funnel_1 THEN
				fbEventButton(eventClass := TC_EVENTS.Entobel.Event177.uuidEventClass, nEventID := 177,
							  sString := REAL_TO_STRING(PR_Line02.fSlow_Speed_vibrating_funnel_1)); 
				nstatechange := 0;
			ELSIF fSlow_Speed_vibrating_funnel_2_line2_change <> PR_Line02.fSlow_Speed_vibrating_funnel_2 THEN
				fbEventButton(eventClass := TC_EVENTS.Entobel.Event178.uuidEventClass, nEventID := 178,
							  sString := REAL_TO_STRING(PR_Line02.fSlow_Speed_vibrating_funnel_2)); 
				nstatechange := 0;
			ELSIF fDerisedWeight_Worm_line2_change <> PR_Line02.fDerisedWeight_Worm THEN
				fbEventButton(eventClass := TC_EVENTS.Entobel.Event179.uuidEventClass, nEventID := 179,
							  sString := REAL_TO_STRING(PR_Line02.fDerisedWeight_Worm)); 
				nstatechange := 0;
			ELSIF fChangeMode_Worm_1_line2_change <> PR_Line02.fChangeMode_Worm_1 THEN
				fbEventButton(eventClass := TC_EVENTS.Entobel.Event180.uuidEventClass, nEventID := 180,
							  sString := REAL_TO_STRING(PR_Line02.fChangeMode_Worm_1)); 
				nstatechange := 0;
			ELSIF fChangeMode_Worm_2_line2_change <> PR_Line02.fChangeMode_Worm_2 THEN
				fbEventButton(eventClass := TC_EVENTS.Entobel.Event181.uuidEventClass, nEventID := 181,
							  sString := REAL_TO_STRING(PR_Line02.fChangeMode_Worm_2)); 
				nstatechange := 0;
			ELSIF fPerStop_Worm_line2_change <> PR_Line02.fPerStop_Worm THEN
				fbEventButton(eventClass := TC_EVENTS.Entobel.Event182.uuidEventClass, nEventID := 182,
							  sString := REAL_TO_STRING(PR_Line02.fPerStop_Worm)); 
				nstatechange := 0;
			ELSIF fTimer_Check_Worm_line2_change <> PR_Line02.fTimer_Check_Worm THEN
				fbEventButton(eventClass := TC_EVENTS.Entobel.Event183.uuidEventClass, nEventID := 183,
							  sString := REAL_TO_STRING(PR_Line02.fTimer_Check_Worm)); 
				nstatechange := 0;
			ELSIF fDelta_Worm_line2_change <> PR_Line02.fDelta_Worm THEN
				fbEventButton(eventClass := TC_EVENTS.Entobel.Event184.uuidEventClass, nEventID := 184,
							  sString := REAL_TO_STRING(PR_Line02.fDelta_Worm)); 
				nstatechange := 0;
			END_IF
	END_CASE
END_IF
END_ACTION

ACTION Reset_active:
PR_Line01.Reset();
END_ACTION

ACTION Start_active:
PR_Conveyor_Out.Stop();
END_ACTION

ACTION steCyclic_active:
PR_Line01();
PR_Conveyor_Out();
MapRtig();
ListError();
PRG_MainRecipe1();
GetLocalSystemTime(bEnable := 1,);
SystemTimeFull 	:= SYSTEMTIME_TO_STRING(in := GetLocalSystemTime.systemTime);
Onlyday 	:= MID(STR:= SystemTimeFull, LEN:=10 , POS:=1 );
OnlyTime 	:= MID(STR:= SystemTimeFull, LEN:=8 , POS:=12 );
//login
IF username <> '' THEN
	openstartpage := TRUE;
ELSE
	openstartpage := FALSE;
END_IF
getuser := WSTRING_TO_STRING(VisuElems.CurrentUserGroupName);

IF VisuElems.CURRENTLANGUAGE = 'vn' THEN
	GVL_OF_VU.bVN := TRUE;
ELSE
	GVL_OF_VU.bVN := FALSE;
END_IF

IF NOT bEmer THEN
	PR_Conveyor_Out.Stop();
	traError := TRUE;
	bLight_Running := FALSE;
	bLight_Stop := TRUE;
END_IF

IF bError1 THEN 
	traError := TRUE;
END_IF

Run_conveyor(CLK := bStart);
Stop_conveyor(CLK := bStop);
IF Run_conveyor.Q THEN
	status := 'RUN';
	bRun := TRUE;
	bStopConv := FALSE;
END_IF

IF bReset THEN
	bWarning := FALSE;
END_IF

IF Stop_conveyor.Q THEN
	bStopConv := TRUE;
	bRun := FALSE;
END_IF

IF bStart THEN
	bfinish1 := TRUE;
	bfinish2 := TRUE;
END_IF

IF bRun THEN
	PR_Conveyor_Out.Auto();
	bLight_Running := TRUE;
	bLight_Stop	:= FALSE;
ELSIF bStopConv AND bfinish1 AND bfinish2 THEN
	PR_Conveyor_Out.Stop();
	status := 'STOP';
	bRun := FALSE;
	bLight_Running := FALSE;
	bLight_Stop	:= TRUE;
END_IF

CASE nWriteData OF 
	0:
		TimerData(IN := TRUE, PT := T#0.5S);
		WritePSData(NETID:='', PORT:=851, START:=FALSE, TMOUT:=T#1S );
		IF TimerData.Q THEN
			nWriteData := 1;
		END_IF
	1:
		TimerData(IN := FALSE);
		nWriteData := 2;
	2:
		TimerData(IN := TRUE, PT := T#0.5S);
		WritePSData(NETID:='', PORT:=851, START:= TRUE, TMOUT:=T#1S );
		IF TimerData.Q THEN
			nWriteData := 3;
		END_IF
	3:
		TimerData(IN := FALSE);
		nWriteData := 0;
END_CASE

IF PR_Conveyor_Out.fb_Conveyor.fbInverter.bVFD THEN
	bRunAuto := TRUE;
ELSE
	bRunAuto := false;
END_IF

CASE nState_IoT OF
	0:
		IF bAlarm THEN
			nState_IoT := 1;
		ELSE
			fbTimer_IoT(IN := TRUE, PT := T#10S);
			IF fbTimer_IoT.Q THEN
				F_SetWarning(115,1);
				F_SetWarning(115,2);
				nState_IoT := 2;
			END_IF
		END_IF
	1:
		bAlarm := FALSE;
		fbTimer_IoT(IN := FALSE);
		nState_IoT := 0;
	2:
		fbTimer_IoT(IN := FALSE);
		IF bAlarm OR bReset THEN
			bWrn := FALSE;
			bWrn2 := FALSE;
			bAlarm_Iot := FALSE;
			nState_IoT := 0;
			bSirens := FALSE;
		END_IF
END_CASE
//Error List
IF bWriteAlarm THEN
FOR k1 := 1 TO 100 DO
	AlarmList[1,k1] 	:= INT_TO_WSTRING(nErrorIDList1[k1].nErrorID);
	AlarmList3[1,k1]	:= INT_TO_STRING(nErrorIDList1[k1].nErrorID);
	AlarmList[4,k1] 	:= STRING_TO_WSTRING(MID(STR := DT_TO_STRING(nErrorIDList1[k1].ErrorTime),LEN := 19, POS := 4));
	AlarmList3[4,k1] 	:= MID(STR := DT_TO_STRING(nErrorIDList1[k1].ErrorTime),LEN := 19, POS := 4);
	IF nErrorIDList1[k1].ErrorStatus = 1 THEN
		AlarmList[3,k1] := "Active";
		AlarmList3[3,k1] := 'Active';
	ELSE
		AlarmList[3,k1] := "Release";
		AlarmList3[3,k1] := 'Release';
	END_IF
	CASE nErrorIDList1[k1].nErrorID OF
			0: 
				AlarmList[4,k1] := "";
				AlarmList[3,k1] := "";
				AlarmList3[4,k1] := '';
				AlarmList3[3,k1] := '';
			1:
				AlarmList[2,k1]  := "E1_1.Lỗi hết hũ trạm 1 [kiểm tra U1I5-2]";
				AlarmList3[2,k1] := 'E1_1.The jar is empty line 1 [check U1I5-2]';
			2:
				AlarmList[2,k1] := "E2_1.Lỗi hũ bị kẹt trạm 1 [kiểm tra U1I5-6]";
				AlarmList3[2,k1] := 'E2_1.The jar  is trapped line 1 [check U1I5-6]';
			3:
				AlarmList[2,k1] := "E3_1.Lỗi ben chặn hũ trên rút về trạm 1 [kiểm tra U1I5-3]" ;
				AlarmList3[2,k1] := 'E3_1.The upper cylinder retract  is faulty line 1 [check U1I5-3]';
			4:
				AlarmList[2,k1] := "E4_1.Lỗi ben chặn hũ dưới rút về trạm 1 [kiểm tra U1I5-4]";
				AlarmList3[2,k1] := 'E4_1.The lower cylinder retract  is faulty line 1 [check U1I5-4]';
			5:
				AlarmList[2,k1] := "E5_1.Lỗi ben chặn hũ dưới đẩy ra trạm 1 [kiểmtra U1I5-5]";
				AlarmList3[2,k1] := 'E5_1.The lower cylinder extend  is faulty line 1 [check U1I5-5]';
			6:
				AlarmList[2,k1] := "E6_1.Lỗi biến tần đảo thức ăn trạm 1 [kiểm tra biến tần 4]";
				AlarmList3[2,k1] := 'E6_1.The inverter of agitator motor fault line 1 [check U1I5-6]';
			7:
				AlarmList[2,k1] := "E7_1.Lỗi driver chia thức ăn trạm 1 [kiểm tra driver 2]";
				AlarmList3[2,k1] := 'E7_1.The driver of dispenser motor fault line 1 [check driver 2]';
			8:
				AlarmList[2,k1] := "E8_1.Lỗi ben chặn sâu rút về trạm 1 [kiểm tra U1I5-7]";
				AlarmList3[2,k1] := 'E8_1.The cylinder blocking worm retract  is faulty line 1 [check U1I5-7]';
			9:
				AlarmList[2,k1] := "E9_1.Lỗi biến tần phểu rung sâu trạm 1 [kiểm tra biến tần 5]";
				AlarmList3[2,k1] := 'E9_1.The inverter of vibrating funnel fault line 1 [check inverter 5]';
			10:
				AlarmList[2,k1] := "E10_1.Lỗi hết nắp trạm 1 [kiểm tra U1I5-8]";
				AlarmList3[2,k1] := 'E10_1.The lid is empty line 1 [check U1I5-8]';
			11:
				AlarmList[2,k1] := "E11_1.Lỗi ben chặn nắp rút về trạm 1 [kiểm tra U1I6-1]";
				AlarmList3[2,k1] := 'E11_1.The cylinder blocking the lid retract is faulty line 1 [check U1I6-1]';
			12:
				AlarmList[2,k1] := "E12-1.Lỗi ben chặn nắp đẩy ra trạm 1 [kiểm tra U1I6-2]";
				AlarmList3[2,k1] := 'E12_1.The cylinder blocking the lid extend is faulty line 1 [check U1I6-2]';
			13:
				AlarmList[2,k1] := "E13_1.Lỗi ben hút/thả nắp rút về trạm 1 [kiểm tra U1I6-3]";
				AlarmList3[2,k1] := 'E13_1.The cylinder sucking the lid retract is faulty line 1 [check U1I6-3]';
			14:
				AlarmList[2,k1] := "E14_1.Lỗi ben hút/thả nắp đẩy ra trạm 1 [kiểm tra U1I6-4]";
				AlarmList3[2,k1] := 'E14_1.The cylinder sucking the lid extend is faulty line 1 [check U1I6-4]';
			15:
				AlarmList[2,k1] := "E15_1.Lỗi ben dập nắp rút về trạm 1 [kiểm tra U1I6-6]";
				AlarmList3[2,k1] := 'E15_1.The cylinder pressing the lid retract is faulty line 1 [check U1I6-6]';
			16:
				AlarmList[2,k1] := "E16_1.Lỗi ben dập nắp đẩy ra trạm 1 [kiểm tra U1I6-7]";
				AlarmList3[2,k1] := 'E16_1.The cylinder pressing the lid extend is faulty line 1 [check U1I6-7]';
			17:
				AlarmList[2,k1] := "E17_1.Lỗi ben lượt ra/vào rút về trạm 1 [kiểm tra U1I6-8]";
				AlarmList3[2,k1] := 'E17_1.The comb cylinder retract is faulty line 1 [check U1I6-8]';
			18:
				AlarmList[2,k1] := "E18_1.Lỗi ben lượt ra/vào đẩy ra trạm 1 [kiểm tra U1I7-1]";
				AlarmList3[2,k1] := 'E18_1.The comb cylinder extend is faulty line 1 [check U1I7-1]';
			19:
				AlarmList[2,k1] := "E19_1.Lỗi ben kẹp hũ rút về trạm 1 [kiểm tra U1I7-4]";
				AlarmList3[2,k1] := 'E19_1.The clap cylinder retract is faulty line 1 [check U1I7-4]';
			20:
				AlarmList[2,k1] := "E20_1.Lỗi ben kẹp hũ đẩy ra trạm 1 [kiểm tra U1I7-5]";	
				AlarmList3[2,k1] := 'E20_1.The clap cylinder extend is faulty line 1 [check U1I7-5]';
			21:
				AlarmList[2,k1] := "E21_1.Lỗi ben di chuyển lượt rút về trạm 1 [kiểm tra U1I7-2]";	
				AlarmList3[2,k1] := 'E21_1.The cylinder moving comb retract is faulty line 1 [check U1I7-2]';
			22:
				AlarmList[2,k1] := "E22_1.Lỗi ben di chuyển lượt đẩy ra trạm 1 [kiểm tra U1I7-3]";
				AlarmList3[2,k1] := 'E22_1.The cylinder moving comb extend is faulty line 1 [check U1I7-3]';
			45:
				AlarmList[2,k1] := "E23_1.Lỗi mất hũ khi đang cân thức ăn trạm 1 [kiểm tra U1I7-6]";
				AlarmList3[2,k1] := 'E23_1.The jar is missed when weighting food line 1 [check U1I7-6]';
			47:
				AlarmList[2,k1] := "E24_1.Lỗi mất hũ khi đang cân sâu trạm 1 [kiểm tra U1I7-7]";
				AlarmList3[2,k1] := 'E24_1.The jar is missed when weighting larvae line 1 [check U1I7-7]';
			49:
				AlarmList[2,k1] := "E25_1.Lỗi hút không được nắp trạm 1 [kiểm tra U1I6-5]";
				AlarmList3[2,k1] := 'E25_1.Failed to suction the lid line 1 [check U1I6-5]';
			51:
				AlarmList[2,k1] := "E26_1.Lỗi nắp đã được hút trạm 1 [kiểm tra U1I6-5]";
				AlarmList3[2,k1] := 'E26_1.The lid is still on the valve line 1 [check U1I5-6]';
			53:
				AlarmList[2,k1] := "E27_1.Lỗi an toàn cửa 1 [kiểm tra U1I7-8]";	
				AlarmList3[2,k1] := 'E27_1.The safety door 1 is error [check U1I7-8]';
			54:
				AlarmList[2,k1] := "E28_1.Lỗi an toàn cửa 2 [kiểm tra U1I7-9]";
				AlarmList3[2,k1] := 'E28_1.The safety door 2 is error [check U1I7-9]';
			55:
				AlarmList[2,k1] := "E29_1.Lỗi an toàn cửa 3 [kiểm tra U1I7-10]";
				AlarmList3[2,k1] := 'E29_1.The safety door 3 is error [check U1I7-10]';
			56: 
				AlarmList[2,k1] := "E30_1.Lỗi quá cân thức ăn trạm 1 [kiểm tra cân thức ăn]";
				AlarmList3[2,k1] := 'E30_1.Overload weightfood [check U1I5-6]';
			57: 
				AlarmList[2,k1] := "E31_1.Lỗi quá cân sâu trạm 1 [kiểm tra cân sâu]";
				AlarmList3[2,k1] := 'E30_1.Overload weightLarvae [check U1I5-6]';	
			60:
				AlarmList[2,k1] := "E32_1.Lỗi ben hút/thả hũ đẩy ra trạm 1 [kiểm tra U1I7-11]";
				AlarmList3[2,k1] := 'E32_1.The cylinder sucking the jar is faulty line 1 [check U1I7-11]'; 
			64:
				AlarmList[2,k1] := "E33_1.Lỗi Modbus thiết bị 3";
				AlarmList3[2,k1] := 'E33_1.Error Modbus device 3';	
			65:
				AlarmList[2,k1] := "E34_1.Lỗi Modbus thiết bị 4";
				AlarmList3[2,k1] := 'E34_1.Error Modbus device 4';
			66:
				AlarmList[2,k1] := "E35_1.Lỗi Modbus thiết bị 5";
				AlarmList3[2,k1] := 'E35_1.Error Modbus device 5';	
			68:
				AlarmList[2,k1] := "E36_1.Lỗi Modbus thiết bị 7";
				AlarmList3[2,k1] := 'E36_1.Error Modbus device 7';	
			69:
				AlarmList[2,k1] := "E37_1.Lỗi đầu cân thức ăn Mettler Toledo 1";
				AlarmList3[2,k1] := 'E37_1.Error Mettler Toledo 1';	
			70:
				AlarmList[2,k1] := "E38_1.Lỗi đầu cân sâu Mettler Toledo 2";
				AlarmList3[2,k1] := 'E38_1.Error Mettler Toledo 2';
			73:
				AlarmList[2,k1] := "E39_1.Lỗi ben chặn sâu đẩy ra trạm 1 [kiểm tra U1I5-7]";
				AlarmList3[2,k1] := 'E39_1.The cylinder blocking worm extend  is faulty line 1';	
			75:
				AlarmList[2,k1] := "E40_1.Lỗi thiếu khí đầu vào [kiểm tra U1I7-13]";
				AlarmList3[2,k1] := 'E40_1.Error of lack of input air [check U1I7-13]';	
			76:
				AlarmList[2,k1] := "E41_1.Lỗi hết thức ăn trạm 1";
				AlarmList3[2,k1] := 'E41_1.Error running out of food line 1';
			77:
				AlarmList[2,k1] := "E42_1.Lỗi hết sâu trạm 1";
				AlarmList3[2,k1] := 'E42_1.Error running out of larvae line 1';		
			98:
				AlarmList[2,k1] := "E98_1.Dừng khẩn [kiểm tra Emergency]";
				AlarmList3[2,k1] := 'E98_1.Emergency Stop [check Emergency]';	 
			99: 
				AlarmList[2,k1] := "E99_1.Lỗi biến tần băng tải đầu ra [kiểm tra biến tần 3]";
				AlarmList3[2,k1] := 'E99_1.The inverter of conveyor out [check inverter 3]';
			101:
				AlarmList[2,k1] := "W1_1.Cảnh báo hết hũ trạm 1[kiểm tra U1I5-2]";
				AlarmList3[2,k1] := 'W1_1.Warning out of jar line 1 [check U1I5-2]';
			102:
				AlarmList[2,k1] := "W2_1.Cảnh báo hết nắp trạm 1[kiểm tra U1I5-8]";
				AlarmList3[2,k1] := 'W2_1.Warning out of lid line 1 [check U1I5-8]';
			103:
				AlarmList[2,k1] := "W3_1.Cảnh báo hết thức ăn trạm 1";
				AlarmList3[2,k1] := 'W3_1.Warning running out of food line 1';
			104:
				AlarmList[2,k1] := "W4_1.Cảnh báo cân quá khối lượng thức ăn trạm 1";
				AlarmList3[2,k1] := 'W4_1.Warning food weight exceeds limit line 1';
			105:
				AlarmList[2,k1] := "W5_1.Cảnh báo hết sâu trạm 1";
				AlarmList3[2,k1] := 'W5_1.Warning running out of larvae line 1';
			106:
				AlarmList[2,k1] := "W6_1.Canh bao can qua khoi luong sau tram 1";
				AlarmList3[2,k1] := 'W6_1.Warning larvae weight exceeds limit line 1';
			107:
				AlarmList[2,k1] := "W7_1.Cảnh báo dập nắp không vô trạm 1[kiểm tra U1I6-7]";
				AlarmList3[2,k1] := 'W7_1.Warning do not press lid inward line 1 [check U1I6-7]';
			115:
				AlarmList[2,k1] := "W8_1.Cảnh báo mất kết nối với PC Advantech [kiểm tra PC]";
				AlarmList3[2,k1] := 'W8_1.Warning disconnect to PC Advantech [check PC]';	
	END_CASE
END_FOR
bWriteAlarm	:= FALSE;
END_IF
END_ACTION

ACTION steError_active:
PR_Line01.Stop();
bStatusStart1 := FALSE;
status := 'ERROR';
bfinish1 := TRUE;
IF i > 100 THEN
	i := 100;
END_IF

CASE nState2 OF 
	0:
		Reset_T(clk := bReset);
		IF Reset_T.Q THEN
			nState2 := 1;
		END_IF
	1:
		timerReset(IN := TRUE, PT := T#500MS);
		PR_Line01.Reset();
		IF nErrorIDList1[1].ErrorStatus = 1 THEN
			IF i <> 1 THEN
				FOR	k := i TO 2 BY -1 DO
				nErrorIDList1[k].nErrorID 	 := nErrorIDList1[k-1].nErrorID;
				nErrorIDList1[k].ErrorTime   := nErrorIDList1[k-1].ErrorTime;
				nErrorIDList1[k].ErrorStatus := nErrorIDList1[k-1].ErrorStatus;		
				END_FOR		
			END_IF 
			nState2 := 2;
		ELSE 
			nState2 := 3;
		END_IF
	2:
		bWriteAlarm	:= TRUE;
		timerReset(IN := TRUE, PT := T#500MS);
		PR_Line01.Reset();
		nErrorIDList1[1].nErrorID := nErrorID;
		nErrorIDList1[1].ErrorTime := SYSTEMTIME_TO_DT(GetLocalSystemTime.systemTime);
		nErrorIDList1[1].ErrorStatus := 0;
		i := i + 1;	
		nState2 := 3;
	3:
		timerReset(IN := TRUE, PT := T#500MS);
		PR_Line01.Reset();
		IF timerReset.Q THEN
			nState2 := 4;
		END_IF
	4:
		timerReset(IN := FALSE);
		Reset_T(clk := FALSE);
		traError := FALSE;
		nState2 := 0;
END_CASE

IF bReset THEN
	bError1 := FALSE;
	bWarning := FALSE;
	bLight_Stop := FALSE;
	bSirens := FALSE;
	status := 'STOP';
	Error[4] := FALSE;
	Error[5] := FALSE;
	Error[7] := FALSE;
	Error[3] := FALSE;
END_IF

IF NOT bEmer THEN
	PR_Line01.Init();
	bRun := FALSE;
END_IF

IF bTo_alarm_side THEN
	VisuElems.CURRENTVISU := 'N_Alarm';
	IF VisuElems.CURRENTVISU = 'N_Alarm' THEN
		bTo_alarm_side := FALSE;
	END_IF
END_IF
END_ACTION

ACTION steErrorCheck_active:

END_ACTION

ACTION steInit_active:
traInitDone := TRUE;
bStatusStart1 := FALSE;
END_ACTION

ACTION steModeAuto_active:
PR_Line01.Auto();
bResetmanual1 := TRUE;
IF bReset THEN
	bWarning := FALSE;
	bSirens  := FALSE;
	bAlarm_Iot := FALSE;
	bWrn 	 := FALSE;
END_IF
END_ACTION

ACTION steModeManual_active:
PR_Line01.Manual();
PR_Line01.Check_reset();
END_ACTION

ACTION steModeSel_active:
IF VisuElems.CURRENTVISU = 'MAIN_LINE1' THEN
	bModeAuto := TRUE;
	bModeManual := FALSE;
END_IF

IF VisuElems.CURRENTVISU = 'N_FoodSupply1' OR VisuElems.CURRENTVISU = 'N_JarSupply1' OR VisuElems.CURRENTVISU = 'N_LidPressing1' OR
	VisuElems.CURRENTVISU = 'N_LidSupply1' OR VisuElems.CURRENTVISU = 'N_Tranfer1' OR VisuElems.CURRENTVISU = 'N_WormWeight1' THEN
	bModeAuto := FALSE;
	bModeManual := TRUE;
END_IF
PR_Line01.check();
bLight_Stop := FALSE;

IF bStart1 THEN
	bStart1 := FALSE;
END_IF
END_ACTION

END_PROGRAM

// ---- POUs/Functions/FB_Eventlogger.TcPOU
FUNCTION_BLOCK FB_Eventlogger
VAR_INPUT
	eventClass: GUID;
	nEventID  : UDINT;
//	sString   : STRING;
END_VAR
VAR_OUTPUT
END_VAR
VAR
	fbEventLogger : FB_TcEventLogger;
	fbSourceInfo  : FB_TcSourceInfo;
END_VAR

fbSourceInfo.Clear();
	fbSourceInfo.sName := '';
	fbSourceInfo.nId := 1;	
fbEventLogger.SendMessage(
	eventClass:= eventClass, 
	nEventId:= nEventID, 
	eSeverity:= TcEventSeverity.Error, 
	ipSourceInfo:= fbSourceInfo, 
	nTimeStamp:= 0, 
	ipArguments:= 0);

END_FUNCTION_BLOCK

// ---- POUs/Functions/FB_EventButton.TcPOU
FUNCTION_BLOCK FB_EventButton
VAR_INPUT
	eventClass: GUID;
	nEventID  : UDINT;
	sString   : STRING;
END_VAR
VAR_OUTPUT
END_VAR
VAR
	fbEventLogger : FB_TcEventLogger;
	fbSourceInfo  : FB_TcSourceInfo;
END_VAR

fbSourceInfo.Clear();
	fbSourceInfo.sName := sString;
	fbSourceInfo.nId := 1;	
fbEventLogger.SendMessage(
	eventClass:= eventClass, 
	nEventId:= nEventID, 
	eSeverity:= TcEventSeverity.Info, 
	ipSourceInfo:= fbSourceInfo, 
	nTimeStamp:= 0, 
	ipArguments:= 0);

END_FUNCTION_BLOCK

// ---- POUs/Functions/F_SetError.TcPOU
FUNCTION F_SetError : BOOL
VAR_INPUT
	nErrID	: INT;
	nLine	: INT;
END_VAR
VAR
END_VAR

IF nLine = 1 THEN
	bError1		:= TRUE;
ELSIF nLine = 2 THEN
	bError2		:= TRUE;
ELSIF nLine = 3 THEN
	bError1		:= TRUE;
	bError2		:= TRUE;
END_IF
nErrorID	:= nErrID;

END_FUNCTION

// ---- POUs/Machines/PR_Conveyor_Out.TcPOU
PROGRAM PR_Conveyor_Out
VAR
	fSpeed_Conveyor			: REAL := 25;
	bUp_Speed				: BOOL;
	bDw_Speed				: BOOL;
	bMotor_Conveyor			: BOOL;
	fb_Conveyor				: FB_FoodMixerModule;
END_VAR

fb_Conveyor(nLine:= 3, UnitID:= 3, fSpeed_motor_mixer:= fSpeed_Conveyor);

ACTION Auto:
fb_Conveyor.Auto();
END_ACTION

ACTION Manual:
fb_Conveyor.Manual(bUp_Motor_Mixer := bUp_Speed, bDown_Motor_Mixer := bDw_Speed,
					bMotor_mixer_Manual := bMotor_Conveyor,bMotor_mixer_reverse := FALSE);
IF bUp_Speed THEN
	bUp_Speed := FALSE;
END_IF

IF bDw_Speed THEN
	bDw_Speed := FALSE;
END_IF
END_ACTION

ACTION Reset:
fb_Conveyor.Reset();
END_ACTION

ACTION Stop:
bMotor_Conveyor		:= FALSE;
fb_Conveyor.Stop();
END_ACTION

END_PROGRAM

// ---- POUs/Components/Child Components/FB_Conveyor.TcPOU
FUNCTION_BLOCK FB_Conveyor IMPLEMENTS I_Conveyor
VAR_INPUT
END_VAR
VAR_OUTPUT
END_VAR
VAR
	//fbInverter		: FB_Inverter;
	bRunConveyor AT %Q* : BOOL;
	bIsRun		 AT %I* : BOOL;
END_VAR

PROPERTY IsRun : BOOL
GET
IsRun := bIsRun;
END_GET
END_PROPERTY

METHOD Start : BOOL
VAR_INPUT
END_VAR
bRunConveyor := TRUE;
END_METHOD

METHOD Stop : BOOL
VAR_INPUT
END_VAR
bRunConveyor := FALSE;
END_METHOD

END_FUNCTION_BLOCK

// ---- POUs/Modules/FB_FoodMixerModule.TcPOU
FUNCTION_BLOCK FB_FoodMixerModule
VAR_INPUT
	nLine				: INT;
	UnitID				: BYTE;
	fSpeed_motor_mixer	: REAL;
	fTimer_Reverse		: REAL;
END_VAR
VAR_OUTPUT
END_VAR
VAR 
	fSpeed_motor_mixer_Manual 		: REAL := 20;
	// ===== CHILD COMPONENTS ======
	fbInverter 			: FB_Inverter;
	// ===== SIM COMPONENTS ======
	fbInverterSim		: FB_Inverter_Sim;
	// ===== INTERFACES ======
	iInverter			: I_Inverter;
	// ======= VAR METHOD =================
	nState							: INT :=0;	
	nStateErr						: INT :=0;
	fbTimer_Err						: TON;
	fbTimer_Reverse					: TON;
	//======= VAR IO =====================
	bError_Motor_Mixer 		AT %I*	: BOOL;
	//========= Var HMI==================
		
END_VAR

IF bSimMode THEN
	iInverter := fbInverterSim;
	fbInverterSim();
ELSE
	iInverter := fbInverter;
	fbInverter(UnitID := UnitID, id := 1);
END_IF

METHOD Auto : BOOL
VAR_INPUT
END_VAR
IF bIsError_Inverter THEN
	IF nLine = 1 THEN
		F_SetError(6,nLine := 1);
	ELSIF nLine = 2 THEN
		F_SetError(28,nLine := 2);
	ELSIF nLine = 3 THEN
		F_SetError(99,nLine := 3);
		bRun := FALSE;
	END_IF
END_IF

IF nLine = 3 THEN
	iInverter.fTargetSpeed	:= fSpeed_motor_mixer;
	iInverter.Start();
ELSE
	CASE nState OF 
		0:
			iInverter.fTargetSpeed	:= fSpeed_motor_mixer;
			iInverter.Start();
			fbTimer_Reverse(IN := TRUE, PT := REAL_TO_TIME(fTimer_Reverse*1000));
			IF fbTimer_Reverse.Q THEN
				nState := 1;
			END_IF
		1:
			fbTimer_Reverse(IN := FALSE);
			iInverter.Stop();
			nState := 2;
		2:
			iInverter.Reverse();
			fbTimer_Reverse(IN := TRUE, PT := REAL_TO_TIME(fTimer_Reverse*1000));
			IF fbTimer_Reverse.Q THEN
				nState := 3;
			END_IF
		3:
			fbTimer_Reverse(IN := FALSE);
			iInverter.Stop();
			nState := 0;
	END_CASE
END_IF
END_METHOD

PROPERTY bIsError_Inverter : BOOL
GET
bIsError_Inverter := bError_Motor_Mixer;
END_GET
END_PROPERTY

METHOD Manual : BOOL
VAR_INPUT
	bUp_Motor_Mixer			: BOOL;
	bDown_Motor_Mixer		: BOOL;
	bMotor_mixer_Manual		: BOOL;
	bMotor_mixer_reverse	: BOOL;
END_VAR
IF bUp_Motor_Mixer THEN
	fSpeed_motor_mixer_Manual	:= fSpeed_motor_mixer_Manual + 0.5;
END_IF

IF bDown_Motor_Mixer THEN
	fSpeed_motor_mixer_Manual 	:= fSpeed_motor_mixer_Manual - 0.5;
END_IF

IF bMotor_mixer_Manual THEN
	iInverter.Start();
ELSIF bMotor_mixer_reverse THEN
	iInverter.Reverse();
ELSIF NOT bMotor_mixer_Manual AND NOT bMotor_mixer_reverse THEN
	iInverter.Stop();
END_IF


iInverter.fTargetSpeed 		:= fSpeed_motor_mixer_Manual;

IF bIsError_Inverter THEN
	IF nLine = 1 THEN
		F_SetError(6,nLine := 1);
	ELSIF nLine = 2 THEN
		F_SetError(28,nLine := 2);
	ELSIF nLine = 3 THEN
		F_SetError(99,nLine := 3);
		iInverter.Stop();
	END_IF
END_IF
END_METHOD

METHOD Reset : BOOL
VAR_INPUT
END_VAR
iInverter.Reset();
fbTimer_Err(IN := false);
END_METHOD

METHOD Stop : BOOL
VAR_INPUT
END_VAR
iInverter.Stop();
nState := 0;
fbTimer_Err(IN := false);
END_METHOD

END_FUNCTION_BLOCK

// ---- POUs/Components/Child Components/FB_Inverter.TcPOU
FUNCTION_BLOCK FB_Inverter IMPLEMENTS I_Inverter
VAR_INPUT
	UnitID		: BYTE;	
	id			: UINT;
END_VAR
VAR_OUTPUT
END_VAR
VAR
	TargetSpeed			: REAL;
	fActualSpeed AT %I*	: REAL;
	bBrake 		 AT %Q* : BOOL;
	bVFD		 AT %Q* : BOOL;
	bReverse	 AT %Q* : BOOL;
	bReset		 AT %Q*	: BOOL;
	nErrId				: INT;
	
	fbInterfaceMbus		: FB_Interface_MbRtu;
	bExecute 			: BOOL;
	bStop				: BOOL;
	WriteVal1			: REAL;
	WriteVal2			: REAL;
	WriteVal3			: REAL;
END_VAR

fbInterfaceMbus(
	UnitID:= UnitID, 
	bExecute:= bExecute, 
	bStop:= bStop, 
	bReset:= bReset,
	idDevice := id,
	fTargetSpeed:= fTargetSpeed);

PROPERTY ActualSpeed : REAL
GET
ActualSpeed := fActualSpeed/100;
END_GET
END_PROPERTY

PROPERTY bIsMove : BOOL
GET
IF bVFD OR bReverse THEN 
	bIsMove := TRUE;
ELSIF NOT bVFD AND NOT bReverse THEN
	bIsMove := FALSE;
END_IF
END_GET
END_PROPERTY

PROPERTY fTargetSpeed : REAL
GET
fTargetSpeed := TargetSpeed;
END_GET
SET
TargetSpeed := fTargetSpeed;
END_SET
END_PROPERTY

METHOD Reset : BOOL
VAR_INPUT
END_VAR
bStop	 := FALSE;
bReset	 := TRUE;
bExecute := FALSE;
bVFD	 := FALSE;
END_METHOD

METHOD Reverse : BOOL
VAR_INPUT
END_VAR
bExecute := TRUE;
bStop	 := FALSE;
bReset	 := FALSE;
bReverse := TRUE;
bVFD 	 := false;
END_METHOD

METHOD Start : BOOL
VAR_INPUT
END_VAR
bExecute := TRUE;
bStop	 := FALSE;
bReset	 := FALSE;
bVFD	 := TRUE;
bReverse := false;
END_METHOD

METHOD Stop : BOOL
VAR_INPUT
END_VAR
bExecute := FALSE;
bStop	 := TRUE;
bReset	 := FALSE;
bVFD	 := FALSE;
bReverse := false;
END_METHOD

END_FUNCTION_BLOCK

// ---- POUs/Components/Child Components/FB_Interface_MbRtu.TcPOU
FUNCTION_BLOCK FB_Interface_MbRtu
VAR_INPUT
	UnitID			: BYTE;
	bExecute		: BOOL;
	bStop			: BOOL;
	bReset			: BOOL;
	idDevice		: UINT;
	fTargetSpeed	: REAL;
END_VAR
VAR_OUTPUT
END_VAR
VAR
	tmp				: WORD;
	bFB_Stop		: BOOL;
	Address1		: WORD;
	Address2		: WORD;
	Address3		: WORD;
	WriteVal  		: WORD;
	WriteVal2		: ARRAY [1..2] OF WORD;
	nState			: INT;
	fbTimer			: TON;
	nStateAll		: INT;
END_VAR

CASE nStateAll OF
	0:
		t := 1;
		nStateAll := 1;
	1:
		IF UnitID = t THEN
			IF idDevice = 1 THEN
				IF WriteVal <> REAL_TO_WORD(fTargetSpeed*100) THEN
					WriteVal := REAL_TO_WORD(fTargetSpeed*100);
					nStateAll := 2;
				ELSE 
					nStateAll := 9;
				END_IF
			ELSIF idDevice = 2 THEN
				IF WriteVal2[1] <> REAL_TO_WORD(fTargetSpeed) THEN
					WriteVal2[1] := REAL_TO_WORD(fTargetSpeed);
					nStateAll := 3;
				ELSE
					nStateAll := 9;
				END_IF
			END_IF
		END_IF
	2:
		fbTimer(IN := TRUE, PT := T#100MS);
		fbModbus.WriteRegs(
						UnitID:= UnitID, 
						Quantity:= 1, 
						MBAddr:= 8193, 
						cbLength:= SIZEOF(WriteVal), 
						pMemoryAddr:=  ADR(WriteVal), 
						Execute:= TRUE, 
						Timeout:= T#1S, 
						BUSY=> Busy[UnitID], 
						Error=> Error[UnitID], 
						ErrorId=> ErrorID[UnitID] , 
						cbRead=> );
		IF fbTimer.Q AND NOT Busy[UnitID] THEN
			nStateAll := 9;
		END_IF
	3:
		fbTimer(IN := TRUE, PT := T#100MS);
		fbModbus.WriteRegs(
						UnitID:= UnitID, 
						Quantity:= 2, 
						MBAddr:= 1034, 
						cbLength:= SIZEOF(WriteVal2), 
						pMemoryAddr:=  ADR(WriteVal2), 
						Execute:= TRUE, 
						Timeout:= T#1S, 
						BUSY=> Busy[UnitID], 
						Error=> Error[UnitID], 
						ErrorId=> ErrorID[UnitID], 
						cbRead=> );
		IF fbTimer.Q AND NOT Busy[UnitID] THEN
			nStateAll := 9;	
		END_IF			
	9:
		fbTimer(IN := false);
		fbModbus.WriteRegs(Execute := FALSE);
		t := t + 1;
		nStateAll := 11;
	11:
		IF t > 7 THEN
			t := 1;
			nStateAll := 1;
		ELSE
			nStateAll := 1;
		END_IF	
END_CASE

END_FUNCTION_BLOCK

// ---- POUs/Components/Sim Components/FB_Inverter_Sim.TcPOU
FUNCTION_BLOCK FB_Inverter_Sim IMPLEMENTS I_Inverter
VAR_INPUT
END_VAR
VAR_OUTPUT
END_VAR
VAR
	TargetSpeed			: REAL;
	fActualSpeed 		: REAL;
	bBrake 		  		: BOOL;
	nErrId				: INT;
	bExecute 			: BOOL;
	bStop				: BOOL;
	bReset				: BOOL;
	//Var sim
	nState				: INT;
	tTimer				: TON;
	tDelay				: TIME := T#2000MS; //acceleration time of inverter
	bStopInit			: BOOL := TRUE;
	fTargetSpeed_re1	: REAL;
	fTargetSpeed_re2	: REAL;
	fActualSpeed_re		: REAL;
END_VAR

CASE nState OF
	0: //init set stop inverter
		IF bStopInit THEN
			bStop := TRUE;
			fActualSpeed := 0;
			tTimer(IN := FALSE);
		END_IF
		nState := nState + 1;
	1://Inv Stop
		fActualSpeed := 0;
		tTimer(IN := FALSE);
		
	10://Inv Run after bExecute = true and speed <> 0
		tTimer(IN := TRUE,PT := tDelay);
		fActualSpeed := fActualSpeed_re + (TIME_TO_REAL(tTimer.ET)*(fTargetSpeed_re1/TIME_TO_REAL(tDelay)));
		fInvSpeed := fActualSpeed;
		// check when change targetspeed
		IF fTargetSpeed_re2 < fTargetSpeed OR fTargetSpeed_re2 > fTargetSpeed THEN
			nState := 20;
		END_IF
	20:
		fActualSpeed_re := fActualSpeed;
		fTargetSpeed_re1 := fTargetSpeed - fActualSpeed;
		fTargetSpeed_re2 := fTargetSpeed;
		tTimer(IN := FALSE);
		nState := 10;
		
END_CASE

//check for signal
IF bExecute AND (fTargetSpeed <> 0) AND (nState = 1) THEN
	fTargetSpeed_re1 := fTargetSpeed;
	fTargetSpeed_re2 := fTargetSpeed;
	fActualSpeed_re := fActualSpeed;
	tTimer(IN := FALSE);
	nState := 10;//Inv run
END_IF

IF bStop THEN
	fActualSpeed := 0;
	nState := 1;//
END_IF

IF fActualSpeed = 0 THEN
	bHaveLoad := FALSE;
ELSE
	bHaveLoad := TRUE;
END_IF

PROPERTY ActualSpeed : REAL
GET
ActualSpeed := fActualSpeed/100;
END_GET
END_PROPERTY

PROPERTY bIsMove : BOOL
GET
IF ActualSpeed > 3 THEN
	bIsMove := FALSE;
ELSE
	bIsMove := TRUE;
END_IF
END_GET
END_PROPERTY

PROPERTY fTargetSpeed : REAL
GET
fTargetSpeed := TargetSpeed;
END_GET
SET
TargetSpeed := fTargetSpeed;
END_SET
END_PROPERTY

METHOD Reset : BOOL
VAR_INPUT
END_VAR
bExecute := FALSE;
bStop	 := FALSE;
bReset	 := TRUE;
END_METHOD

METHOD Reverse : BOOL
VAR_INPUT
END_VAR
END_METHOD

METHOD Start : BOOL
VAR_INPUT
END_VAR
bExecute := TRUE;
bStop	 := FALSE;
bReset	 := FALSE;
END_METHOD

METHOD Stop : BOOL
VAR_INPUT
END_VAR
bExecute := FALSE;
bStop	 := TRUE;
bReset	 := FALSE;
END_METHOD

END_FUNCTION_BLOCK

// ---- POUs/Machines/PR_Line01.TcPOU
PROGRAM PR_Line01
VAR PERSISTENT
//----------------VAR SETTING--------------------
	timerCheckCylinder_Up			: REAL;//CupSupply
	timerCheckCylinder_Dw			: REAL;
	timerCheckEmpty					: REAL;
	timerCheckStuck					: REAL;
	timerCylinder_Up_extend 		: REAL;
	timerCylinder_Suction_Cup_extend: REAL;
	timerCylinder_Suction_Cup		: REAL;
	timerCylinder_Suction_Val		: REAL;
	timerCylinder_Suction_pick		: REAL;
	fSpeed_motor_mixer				: REAL;//FoodMixer
	fTimer_Reverse					: REAL;
	fFast_Speed						: REAL;//FoodWeight
	fSlow_Speed_1					: REAL;
	fSlow_Speed_2					: REAL;
	fDerisedWeight_Food				: REAL;
	fChangeMode_Food_1				: REAL;
	fChangeMode_Food_2				: REAL;
	fMaxWeight_Food					: REAL;
	fPerStop_Food					: REAL;
	fTimer_Food						: REAL;
	fTimer_Alarm_Food				: REAL;
	fTimer_Check_Food				: REAL;
	fDelta_Food						: REAL;
	fTimer_rever_food				: REAL;
	fTimer_Error_Food				: REAL;
	fFast_Speed_vibrating_funnel	: REAL;//WormWeight
	fSlow_Speed_vibrating_funnel_1	: REAL;
	fSlow_Speed_vibrating_funnel_2	: REAL;
	fDerisedWeight_Worm				: REAL;
	fChangeMode_Worm_1				: REAL;
	fChangeMode_Worm_2				: REAL;
	fMaxWeight_Worm					: REAL;
	fPerStop_Worm					: REAL;
	fTimer_Worm						: REAL;
	fTimer_Alarm_Worm				: REAL;
	fTimer_Check_Worm				: REAL;
	fTimer_Check_Cylinder			: REAL;
	fDelta_Worm						: REAL;
	fTimer_Error_Worm				: REAL;
	timerCylinder_Suction			: REAL;//LidSupply
	timerCheckLidRelease			: REAL;
	timerLidBlow					: REAL;
	timerCheckLidEmpty				: REAL;
	timerCheckLidSuck				: REAL;
	timerCylinder_Stopper			: REAL;
	timer_Check_Cylinder_extend		: REAL;//LidClose
	timer_Check_Cylinder_retract	: REAL;
	timer_CloseLid					: REAL;
	fTimer_Comb						: REAL;//Transfer
	fTimer_Clip						: REAL;
	fTimer_Move_Comb				: REAL;
//-----------------VAR HMI-------------------
	fProductLog						: ARRAY [1..2] OF ARRAY  [1..5] OF REAL;
END_VAR

VAR
	bStatus_Food					: BOOL;
	bStatus_Worm					: BOOL;
//----------------VAR MANUAL---------------------
	bCylinder_up_extend 			: BOOL;//CupSupply
	bCylinder_up_retract 			: BOOL;
	bCylinder_dw_extend 			: BOOL;
	bCylinder_dw_retract 			: BOOL;
	bCylinder_Suction_cup_extend	: BOOL;
	bCylinder_Suction_cup_retract	: BOOL;
	bUp_Motor_Mixer					: BOOL;//FoodMixer
	bDown_Motor_Mixer				: BOOL;
	bMotor_mixer_Manual				: BOOL;
	bMotor_mixer_reverse			: BOOL;
	bUp_Food_Motor					: BOOL;//FoodWeight
	bDown_Food_Motor				: BOOL;
	bZero_Loadcell_Food				: BOOL;
	bMotor_Food						: BOOL;
	bMotor_Food_reverse				: BOOL;
	bUp_vibrating_funnel			: BOOL;//WormWeight
	bDown_vibrating_funnel			: BOOL;
	bZero_Loadcell_Worm				: BOOL;
	bCylinder_Block_Worm_Extend		: BOOL;
	bCylinder_Block_Worm_Retract	: BOOL;
	bMotor_vibrating_funnel			: BOOL;	
	bCylinder_LidStopper_extend 	: BOOL;//LidSupply
	bCylinder_LidStopper_retract 	: BOOL;
	bCylinder_Suction_extend		: BOOL;
	bCylinder_Suction_retract		: BOOL;
	bLidSuctionValve				: BOOL;
	bCupSuctionValve				: BOOL;
	bBlowValve						: BOOL;
	bCylinder_CloseLid_Extend		: BOOL;//LidClose
	bCylinder_CloseLid_Retract		: BOOL;
	bCylinder_Comb_Extend			: BOOL;//Transfer
	bCylinder_Comb_Retract			: BOOL;
	bCylinder_Clip_Extend			: BOOL;
	bCylinder_Clip_Retract			: BOOL;
	bCylinder_Move_Comb_Extend		: BOOL;
	bCylinder_Move_Comb_Retract		: BOOL;
//------------------fbmodule----------------
	fb_CupSupply	: FB_CupSupplyModule;
	fb_FoodMixer	: FB_FoodMixerModule;
	fb_FoodWeight	: FB_FoodWeightModule;
	fb_WormWeight	: FB_WormWeightModule;
	fb_LidSupply	: FB_LidSupplyModule;
	fb_LidClose		: FB_LidCloseModule;
	fb_Transfer		: FB_Transfer;
//---------------- VAR Method ---------------
	nState				: INT;
	nState_Dropcup		: INT;
	nState_Transfer		: INT;
	nState_FoodWeight	: INT;
	nState_WormWeight	: INT;
	nState_LidClose		: INT;
	nState_LidSupply	: INT;
	nDoneTransfer		: INT;
	nDoneTransferStop	: INT;
	tmp					: INT;
	bDoneTakeLid		: BOOL;
	bDoneTransfer		: BOOL;
	bDoneCupSupply		: BOOL;
	bDoneFoodWeight		: BOOL;
	bDoneWormWeight		: BOOL;
	bDoneLidSupply		: BOOL;
	bDoneLidClose		: BOOL;
	bEnable				: BOOL;
	bFinishCupSupply	: BOOL;
	bFinishFoodWeight	: BOOL;
	bFinishWormWeight	: BOOL;
	bFinishLidSupply	: BOOL;
	bFinishLidClose		: BOOL;
	bFinishTransfer		: BOOL;
	//-------VAR--------------
	nStateConveyor		: INT;
	fbtimertransfer		: TON;
	nStateStop			: INT;
	fbTimer				: ton;
	fbtimerStop			: ton;
	fbTimerCycle		: ton;
	timeCycle			: REAL :=1;
	fproduct			: INT;
	nstateCycle			: INT;
	bDone				: R_TRIG;
	fbDelay				: TON;
	bStatus_Food_order	: ARRAY [1..3] OF BOOL;
	bStatus_Worm_order	: ARRAY [1..3] OF BOOL;
	bStatus_Lid_order	: ARRAY [1..3] OF BOOL;
	i1,i2,i3			: INT := 0;
	xathucan			: BOOL;
	xasau				: BOOL;
	daothucan			: BOOL;
	transfer			: BOOL;
	nstatetest1			: INT;
	nstatetest2			: INT;
	nstatetest3			: INT;
	nstatetest4         : INT;
	bxa					: BOOL;
	bCheck				: BOOL;
	bypassfood			: BOOL;
	bypassWorm			: BOOL;
	bypassLid			: BOOL;
	eles: INT;
END_VAR

fb_CupSupply(
	nLine:= 1 , 
	timerCheckCylinder_Up:= timerCheckCylinder_Up, 
	timerCheckCylinder_Dw:= timerCheckCylinder_Dw, 
	timerCheckEmpty:= timerCheckEmpty, 
	timerCheckStuck:= timerCheckStuck,
	timerCylinder_Up_extend := timerCylinder_Up_extend,
	timerCylinder_Suction:= timerCylinder_Suction_Cup,
	timerCylinder_Suction_extend:= timerCylinder_Suction_Cup_extend,
	ttimerCylinder_val:= timerCylinder_Suction_Val,
	timerCylinder_Suction_pick:= timerCylinder_Suction_pick);

fb_FoodMixer(
	nLine:= 1,
	UnitID:= 4, 
	fSpeed_motor_mixer:= fSpeed_motor_mixer,
	fTimer_Reverse:= fTimer_Reverse);
		
fb_FoodWeight(
	nLine:= 1, 
	UnitID:= 7, 
	fFast_Speed:= fFast_Speed, 
	fSlow_Speed_1:= fSlow_Speed_1, 
	fSlow_Speed_2:= fSlow_Speed_2, 
	fDerisedWeight_Food:= fDerisedWeight_Food, 
	fChangeMode_Food_1:= fChangeMode_Food_1, 
	fChangeMode_Food_2:= fChangeMode_Food_2, 
	fMaxWeight_Food:= fMaxWeight_Food, 
	fPerStop_Food:= fPerStop_Food, 
	fTimer_Food:= fTimer_Food, 
	fTimer_Alarm_Food:= fTimer_Alarm_Food, 
	fTimer_Check_Food:= fTimer_Check_Food, 
	fDelta_Food:= fDelta_Food,
	fTimer_Reverse := fTimer_rever_food,
	fTimer_Error_Food := fTimer_Error_Food, 
	fProductLogF=> fProductLog[1],
	bStatus_Food=> bStatus_Food,
	Time_start => Time_Start_Food_line1,
	Time_Stop => Time_Stop_Food_line1,
	status=>bStatus_Food_line1,
	fweight_iot =>fWeight_food_line1);

fb_LidClose(
	nLine:= 1, 
	timer_Check_Cylinder_extend:= timer_Check_Cylinder_extend, 
	timer_Check_Cylinder_retract:= timer_Check_Cylinder_retract, 
	timer_CloseLid:= timer_CloseLid);
	
fb_LidSupply(
	nLine:= 1, 
	timerCylinder_Suction:= timerCylinder_Suction, 
	timerCheckLidRelease:= timerCheckLidRelease, 
	timerLidBlow:= timerLidBlow, 
	timerCheckLidEmpty:= timerCheckLidEmpty, 
	timerCheckLidSuck:= timerCheckLidSuck, 
	timerCylinder_Stopper:= timerCylinder_Stopper);

fb_Transfer(
	nLine:= 1, 
	fTimer_Comb:= fTimer_Comb, 
	fTimer_Clip:= fTimer_Clip, 
	fTimer_Move_Comb:= fTimer_Move_Comb, 
	nDoneTransfer=> nDoneTransfer,
	bDoneTransfer=> bDoneTransfer);

